// TwinCAT 3 PLC project MainPLC
// ProgramVersion: 3.1.4026.13
// libraries:
//   Tc2_BA, * (Beckhoff Automation GmbH)
//   Tc2_EtherCAT, * (Beckhoff Automation GmbH)
//   Tc2_Math, * (Beckhoff Automation GmbH)
//   Tc2_Standard, * (Beckhoff Automation GmbH)
//   Tc2_System, * (Beckhoff Automation GmbH)
//   Tc2_Utilities, * (Beckhoff Automation GmbH)
//   Tc3_EventLogger, * (Beckhoff Automation GmbH)
//   Tc3_IotBase, * (Beckhoff Automation GmbH)
// project tree:
//   DUTs/ARDeviceAPI/ keyValuePair_t.TcDUT
//   DUTs/ARDeviceErrorSystemLinker/ ARDeviceErrorSystemLink_t.TcDUT
//   DUTs/ErrorSystem/ ActorMovingTimeoutEx_t.TcDUT, ActorStartMovingtimeoutEx_t.TcDUT, IOExpantionMessageErrorEx_t.TcDUT, PrimitiveWatchdogEx_t.TcDUT
//   DUTs/IOExpantionHandler/ actorID_t.TcDUT, IOExpantionLocation_t.TcTLEO, IOExpantionMessageDescriptor_t.TcDUT, IOExpantionMessageSubData_t.TcDUT, sensorID_t.TcTLEO
//   DUTs/MainStateMachine/ mainStateMachineStatus_t.TcTLEO
//   DUTs/SignalStatusLampTypes/ SignalStatusLampStatus_t.TcTLEO
//   DUTs/systemOperationalTypes/ systemStatus_t.TcTLEO
//   GVLs/ ErrorSystemStatusVar.TcGVL, HMIInterface.TcGVL, InputOutput.TcGVL, test.TcGVL
//   / Klassendiagramm_1.TcCD (not stored), PlcTask.TcTTO
//   POUs/ARCommunication/ ARDeviceAPI_t.TcPOU, ARDeviceErrorSystemLinkerInitialiser.TcPOU, ARDeviceErrorSystemLinker_t.TcPOU
//   POUs/ARCommunication/Helper/ pulseSignalGenerator_t.TcPOU, WSJSONStringBuilder_t.TcPOU
//   POUs/ARCommunication/MQTT/ ARCommunicationMQTTExtention_t.TcPOU, ARCommunicationMQTT_t.TcPOU
//   POUs/ARCommunication/Websocket/ ARCommunicationWSExtentionWS_t.TcPOU, ARCommunicationWS_t.TcPOU
//   POUs/ARUIHandler/ ARUIHandler_t.TcPOU
//   POUs/ErrorSystem/ ActorStartMovingTimeoutManager_t.TcPOU, GernericErrorWatchdog_t.TcPOU, ActorMovingTimeoutManager_t.TcPOU, ErrorManager_t.TcPOU, formatPosition.TcPOU, IOExpantionMessageErrorHandler_t.TcPOU, PrimitiveWatchdogManager_t.TcPOU, SendErrorMessage.TcPOU
//   POUs/HMIHandler/ HMIHandler_t.TcPOU
//   POUs/IOExpantionHandler/ IOExpantionHandler_t.TcPOU
//   POUs/ MAIN.TcPOU
//   POUs/MainStateMachine/ mainStateMachine_t.TcPOU
//   POUs/SignalStatusLamp/ SignalStatusLampComponent_t.TcPOU, SignalStatusLamp_t.TcPOU
// real-time tasks:
//   TASK PlcTask: cycle T#10ms, priority 20, ADS port 350
// I/O:
//   DEVICE Gerät 1 (EtherCAT), AmsNetId 5.85.199.196.2.1
//     Klemme 1 (EK1200) [EK1200-5000 EtherCAT Netzteil (2A E-Bus)]
//       Klemme 2 (EL2869) [EL2869 16K. Dig. Ausgang 24V, 0,5A, Diagnose]
//       Klemme 3 (EL1808) [EL1808 8K. Dig. Eingang 24V, 3ms]
//       Klemme 4 (EL1808) [EL1808 8K. Dig. Eingang 24V, 3ms]
//       Klemme 5 (EL4022) [EL4022 2K. Ana. Ausgang 4-20mA, 12bit]
//       Klemme 6 (EL4104) [EL4104 4Ch. Ana. Ausgang 0-10V, 16bit]
//       Klemme 7 (EL3172) [EL3172 2K. Ana. Eingang +/-10V, +/-20mA, 16 Bit, Galvanisch getrennt]
//       Klemme 8 (EL9011) [EL9011 Endklemme]
//   DEVICE Gerät 3 (EtherCAT), AmsNetId 5.85.199.196.4.1
//     Box 9 (54632) [IMPACT67 Pro EC DIO8 IOL8]
//       modules: Module 1 (Digital_IN), Module 2 (Digital_IN), Module 3 (Digital_IN), Module 4 (Digital_IN), Module 5 (Digital_IN), Module 6 (IOL_0/4_I/O-Bytes), Module 7 (Digital_IN), Module 8 (IOL_4/4_I/O-Bytes)
// variable links:
//   MainPLC/MainPLC Instance <-> Device 1 (EtherCAT)/Term 1 (EK1200)/Term 2 (EL2869)
//     PlcTask Outputs/InputOutput.ConvaorbeltMotorReverse <-> DOS Outputs Channel 7/Output
//     PlcTask Outputs/InputOutput.ConvaorbeltMotorRun <-> DOS Outputs Channel 6/Output
//     PlcTask Outputs/InputOutput.OnOffStatusLamp <-> DOS Outputs Channel 12/Output
//     PlcTask Outputs/InputOutput.QuittierenLamp <-> DOS Outputs Channel 11/Output
//     PlcTask Outputs/InputOutput.TurnTableMotorReverse <-> DOS Outputs Channel 5/Output
//     PlcTask Outputs/InputOutput.TurnTableMotorTurn <-> DOS Outputs Channel 4/Output
//     PlcTask Outputs/MAIN.signalStatusLamp._signalLampGreen._SignalStatusLamp <-> DOS Outputs Channel 3/Output
//     PlcTask Outputs/MAIN.signalStatusLamp._signalLampRed._SignalStatusLamp <-> DOS Outputs Channel 1/Output
//     PlcTask Outputs/MAIN.signalStatusLamp._signalLampYellow._SignalStatusLamp <-> DOS Outputs Channel 2/Output
//   MainPLC/MainPLC Instance <-> Device 1 (EtherCAT)/Term 1 (EK1200)/Term 3 (EL1808)
//     PlcTask Inputs/InputOutput.EmStop <-> Channel 5/Input
//     PlcTask Inputs/InputOutput.ResetButton <-> Channel 6/Input
//   MainPLC/MainPLC Instance <-> Device 1 (EtherCAT)/Term 1 (EK1200)/Term 4 (EL1808)
//     PlcTask Inputs/InputOutput.StartButton <-> Channel 1/Input
//     PlcTask Inputs/InputOutput.StopButton <-> Channel 2/Input
//   MainPLC/MainPLC Instance <-> Device 3 (EtherCAT)/Box 9 (54632)
//     PlcTask Inputs/MAIN.IOExpantionHandler._IOExpantionExpantionInByte_{0..3} <-> Module 8 (IOL_4/4_I/O-Bytes)/TxPDO/input byte {0..3}  (4 links)
//     PlcTask Inputs/MAIN.IOExpantionHandler._IOExpantionIn_0 <-> TxPDO Mapping of Digital Inputs/PD (I/Q Pin2 + C/Q Pin4)
//     PlcTask Outputs/MAIN.IOExpantionHandler._FestoPneumaticOutByte_{0..3} <-> Module 6 (IOL_0/4_I/O-Bytes)/RxPDO/output byte {0..3}  (4 links)

CONFIGURATION MainPLC
    RESOURCE PLC ON TwinCAT3
        TASK PlcTask(INTERVAL := T#10ms, PRIORITY := 20);
        PROGRAM MAIN WITH PlcTask : MAIN;
    END_RESOURCE
END_CONFIGURATION

// ---- DUTs/ARDeviceAPI/keyValuePair_t.TcDUT
TYPE keyValuePair_t :
STRUCT
	key : STRING(255);
	value : string(255);
END_STRUCT
END_TYPE

// ---- DUTs/ARDeviceErrorSystemLinker/ARDeviceErrorSystemLink_t.TcDUT
TYPE ARDeviceErrorSystemLink_t :
STRUCT
	stEventEntity : TcEventEntry;
	callBackPtr : POINTER to bool;
END_STRUCT
END_TYPE

// ---- DUTs/ErrorSystem/ActorMovingTimeoutEx_t.TcDUT
// tis is a class that is used by the ActorMovingTimeoutManager
TYPE ActorMovingTimeoutEx_t :
STRUCT
	ActorMovingTimeout : GernericErrorWatchdog_t;
	sensorPtr1 : POINTER TO BOOL := NULL;
	sensorPtr2 : POINTER TO BOOL := NULL;
	sensorPtr3 : POINTER TO BOOL := NULL;
	sensorID1 : sensorID_t := sensorID_t.SENSOR_NO_SENSOR;
	sensorID2 : sensorID_t := sensorID_t.SENSOR_NO_SENSOR;
	sensorID3 : sensorID_t := sensorID_t.SENSOR_NO_SENSOR;
END_STRUCT
END_TYPE

// ---- DUTs/ErrorSystem/ActorStartMovingtimeoutEx_t.TcDUT
TYPE ActorStartMovingtimeoutEx_t :
STRUCT
	ActorStartMovingTimeout : GernericErrorWatchdog_t;
	expectedActorValue : BOOL; // actor value when sensor is true
	sensorPtr : POINTER TO BOOL := NULL;
	actorPtr : POINTER TO BOOL := NULL;
	sensorID : sensorID_t := sensorID_t.SENSOR_NO_SENSOR;
	actorID : actorID_t := actorID_t.ACTOR_NO_ACTOR;
END_STRUCT
END_TYPE

// ---- DUTs/ErrorSystem/IOExpantionMessageErrorEx_t.TcDUT
TYPE IOExpantionMessageErrorEx_t :
STRUCT
	isErrorActive : BOOL := FALSE; // a variable to attach to primitiveWatchdogHandler
	errorMessageCallback : BOOL := FALSE; // callback for IOExpantionHandler_t
	clearMessageCallback : BOOL := FALSE; // callback for IOExpantionHandler_t
END_STRUCT
END_TYPE

// ---- DUTs/ErrorSystem/PrimitiveWatchdogEx_t.TcDUT
TYPE PrimitiveWatchdogEx_t :
STRUCT
	primitiveWatchdog : GernericErrorWatchdog_t;
	invert : BOOL := FALSE; // if true, inverts the watchdog feeding signal
	sensorID : sensorID_t := sensorID_t.SENSOR_NO_SENSOR;
	sensorPtr : POINTER TO BOOL := NULL;
END_STRUCT
END_TYPE

// ---- DUTs/IOExpantionHandler/actorID_t.TcDUT
{attribute 'qualified_only'}
{attribute 'strict'}
{attribute 'to_string'}
TYPE actorID_t :
(
	ACTOR_0 := 0,
	ACTOR_1,
	ACTOR_2,
	ACTOR_3,
	ACTOR_GRIPPER_RIGHT_LEFT,
	ACTOR_GRIPPER_OPEN_CLOSE,
	ACTOR_GRIPPER_UP_DOWN,
	ACTOR_Y1_OUT,
	ACTOR_Y2_OUT,
	ACTOR_Y3_OUT,
	ACTOR_NO_ACTOR
);
END_TYPE

// ---- DUTs/IOExpantionHandler/IOExpantionLocation_t.TcTLEO
{attribute 'qualified_only'}
{attribute 'strict'}
{attribute 'to_string'}
TYPE IOExpantionLocation_t :
( 
	ROOT := 0, // this is the main IO master
	EXPANTION  // this is the expantion of the IO master
);
END_TYPE

// ---- DUTs/IOExpantionHandler/IOExpantionMessageDescriptor_t.TcDUT
TYPE IOExpantionMessageDescriptor_t :
STRUCT
	diagCode : ARRAY [0..3] OF BYTE;
	textID : ARRAY [0..1] OF BYTE;
END_STRUCT
END_TYPE

// ---- DUTs/IOExpantionHandler/IOExpantionMessageSubData_t.TcDUT
TYPE IOExpantionMessageSubData_t :
STRUCT
	callbackVariable : POINTER TO BOOL := NULL;
	messageDescription : IOExpantionMessageDescriptor_t;
END_STRUCT
END_TYPE

// ---- DUTs/IOExpantionHandler/sensorID_t.TcTLEO
{attribute 'qualified_only'}
{attribute 'strict'}
{attribute 'to_string'}
TYPE sensorID_t :
(
	SENSOR_B8_CONVAYORBELT_METTAL_PRESENT := 0, 
	SENSOR_B5_STORAGE_ENTRANCE,
	
	SENSOR_B17_GRIPPER_RIGHT, 
	SENSOR_B16_GRIPPER_LEFT,
	
	SENSOR_B3_Y3_DOWN, 
	SENSOR_B4_Y3_UP,
	
	EXPANTION_SENSOR_Y4_UP, 
	EXPANTION_SENSOR_B11_Y5_INSIDE,
	
	EXPANTION_SENSOR_B7_ENTRANCE_CONVAYORBELT, 
	EXPANTION_SENSOR_B6_PART_SENSOR_METTAL_PRESENT,
	
	EXPANTION_SENSOR_B12_PART_TURNTABLE_PRESENT, 
	EXPANTION_SENSOR_Y4_DOWN,
	
	EXPANTION_SENSOR_B10_Y5_OUT, 
	EXPANTION_SENSOR_B18_SENSOR_Y4,
	
	EXPANTION_SENSOR_B1_Y2_DOWN, 
	EXPANTION_SENSOR_B2_Y2_UP,
	
	SENSOR_PNEUMATIC_PRESHURE_OK,
	SENSOR_B13_TURNTABLE_POS_REACHED,
	SENSOR_NO_SENSOR
);
END_TYPE

// ---- DUTs/MainStateMachine/mainStateMachineStatus_t.TcTLEO
{attribute 'qualified_only'}
{attribute 'strict'}
{attribute 'to_string'}
TYPE mainStateMachineStatus_t :
(
	IDLE := 0,
	ROTATE_TABLE,
	GRIPPER_DOWN,
	GRIPPER_CLOSE,
	GRIPPER_UP,
	GRIPPER_LEFT,
	GRIPPER_DOWN_LEFT,
	GRIPPER_OPEN,
	GRIPPER_UP_LEFT,
	GRIPPER_RIGHT,
	Y10_OUT,
	CONVAYORBELT_START,
	Y10_BACK,
	Y2_OUT,
	Y3_OUT,
	CONVEYORBELT_STOP
);
END_TYPE

// ---- DUTs/SignalStatusLampTypes/SignalStatusLampStatus_t.TcTLEO
{attribute 'qualified_only'}
{attribute 'strict'}
{attribute 'to_string'}
TYPE SignalStatusLampStatus_t :
(
	NONE := 0,
	OPERATIONAL := 1,
	WARNING := 2,
	ERROR := 3,
	STARTING := 4,
	STOPPING := 5
);
END_TYPE

// ---- DUTs/systemOperationalTypes/systemStatus_t.TcTLEO
{attribute 'qualified_only'}
{attribute 'strict'}
{attribute 'to_string'}
TYPE systemStatus_t :
(
	STOPPED := 0,
	STARTING := 1,
	RUNNING := 2,
	ERROR := 3,
	STOPPING := 4
);
END_TYPE

// ---- GVLs/ErrorSystemStatusVar.TcGVL
{attribute 'qualified_only'}
VAR_GLOBAL
	errorHide_ERR_PNEU_LOW_PR_402 : BOOL := FALSE;
	errorHide_ERR_LD_START_LEFT_408_TIMEOUT : BOOL := FALSE;
	errorHide_ERR_LD_START_RIGHT_408_TIMEOUT : BOOL := FALSE;
	errorHide_ERR_LD_MOVE_408_TIMEOUT : BOOL := FALSE;
	errorHide_ERR_RT_MOVE_408_TIMEOUT : BOOL := FALSE;
	errorHide_ERR_Y2_MOVE_408_TIMEOUT : BOOL := FALSE;
	errorHide_ERR_Y2_START_DOWN_408_TIMEOUT : BOOL := FALSE;
	errorHide_ERR_Y2_START_UP_408_TIMEOUT : BOOL := FALSE;
	errorHide_ERR_Y3_MOVE_408_TIMEOUT : BOOL := FALSE;
	errorHide_ERR_Y3_START_DOWN_408_TIMEOUT : BOOL := FALSE;
	errorHide_ERR_Y3_START_UP_408_TIMEOUT : BOOL := FALSE;
END_VAR

// ---- GVLs/HMIInterface.TcGVL
{attribute 'qualified_only'}
VAR_GLOBAL
	HMIStartStatusLamp : BOOL := FALSE;
	HMIStopStatusLamp : BOOL := FALSE;
	HMIErrorStatusLamp : BOOL := FALSE;
	
	HMIStartMachine : BOOL := FALSE;
	HMIStopMachine : BOOL := FALSE;
END_VAR

// ---- GVLs/InputOutput.TcGVL
{attribute 'qualified_only'}
VAR_GLOBAL
	
	// outputs
	TurnTableMotorTurn AT %Q* : BOOL;
	TurnTableMotorReverse AT %Q* : BOOL;
	ConvaorbeltMotorRun AT %Q* : BOOL;
	ConvaorbeltMotorReverse AT %Q* : BOOL;
	QuittierenLamp AT %Q* : BOOL;
	OnOffStatusLamp AT %Q* : BOOL;

	// inputs
	StartButton AT %I* : BOOL;
	StopButton AT %I* : BOOL;
	EmStop AT %I* : BOOL;
	ResetButton AT %I* : BOOL;
	
	
END_VAR

// ---- GVLs/test.TcGVL
{attribute 'qualified_only'}
VAR_GLOBAL
	testBoolLinker : BOOL := FALSE;
	testBoolLinker2 : BOOL := FALSE;
END_VAR

// ---- POUs/MAIN.TcPOU
PROGRAM MAIN
VAR
signalStatusLamp : SignalStatusLamp_t;

systemStatus : systemStatus_t := systemStatus_t.STOPPED;
ARDevice : ARDeviceAPI_t;

IOExpantionHandler : IOExpantionHandler_t;

mainStateMachine : mainStateMachine_t;

ARUIHandler : ARUIHandler_t;

HMIHandler : HMIHandler_t;

ErrorManager : ErrorManager_t;

ARDeviceErrorSystemLinker : ARDeviceErrorSystemLinker_t;

_ErrorMessage : FB_TcMessage;
_tmpStr : STRING := '';

//test
firstRun : BOOL := FALSE;
run : bool := false;
callback : BOOL := FALSE;

diagCode : ARRAY[0..3] OF BYTE := [16#03, 16#E0, 16#08, 16#00];
textID : ARRAY[0..1] OF BYTE := [16#38, 16#00];

//murr test
	ReadDiag: FB_EcCoESdoRead;
	
BuffDiagMess :Array[0..39] of byte;
	xStart: BOOL;
	ReadLength: UDINT;
END_VAR

IF firstRun = FALSE THEN 
	firstRun := TRUE;
	ARDeviceErrorSystemLinkerInitialiser(ARDeviceErrorSystemLinker, ARDevice);
END_IF


// always update mainStateMachine IOExpantionahndler refferance
mainStateMachine.IOExpantionHandler := ADR(IOExpantionHandler);

ARUIHandler.ARDevice := ADR(ARDevice);
ARUIHandler.systemStatus := ADR(systemStatus);
ARUIHandler.IOExpantionHandler := ADR(IOExpantionHandler);


HMIHandler.systemStatus := ADR(systemStatus);


IF (InputOutput.StartButton OR HMIInterface.HMIStartMachine) AND NOT (systemStatus = systemStatus_t.ERROR) THEN 
	systemStatus := systemStatus_t.RUNNING; // TODO: Starting isn't implemented jet and also isn't really needed at the moment
	//ARCommunication.sendNewMessage(ADR(testStr)); // test for websocet connection
	mainStateMachine.startStateMachine(); // start state machine
	ErrorManager.startErrors();
END_IF
	
IF (NOT InputOutput.StopButton OR HMIInterface.HMIStopMachine) THEN
	mainStateMachine.stopStateMachine(); 
	systemStatus := systemStatus_t.STOPPING; 
END_IF

IF systemStatus = systemStatus_t.STOPPING AND mainStateMachine.getIsStateMachineON() = FALSE THEN
	systemStatus := systemStatus_t.STOPPED; 
	ErrorManager.stopErrors();
END_IF

// push error test
IF (NOT InputOutput.EmStop) AND systemStatus <> systemStatus_t.ERROR AND FALSE THEN 
 			_ErrorMessage.CreateEx(TC_EVENTS.OperationalErrors.EmStopPressed, 0 ); {info 'TODO: make this a alarm and not a message'}
			_ErrorMessage.ipArguments.AddString(__POUNAME());
			_tmpStr := formatPosition(__POSITION());
			_ErrorMessage.ipArguments.AddString(_tmpStr);
			_ErrorMessage.Send(0);
END_IF


IF ErrorManager.hasError() THEN
	// overwrite systemstatus to force to error state
	systemStatus := systemStatus_t.ERROR; 
	mainStateMachine.reset(); // reset StateMachine
	ErrorManager.stopErrors();
END_IF

// reset errors 
IF InputOutput.ResetButton AND systemStatus = systemStatus_t.ERROR THEN
	systemStatus := systemStatus_t.STOPPED;
	ErrorManager.confirmAll();
	InputOutput.QuittierenLamp := FALSE;
END_IF

// set lamp of quittierung
IF ErrorManager.hasError() AND systemStatus = systemStatus_t.ERROR THEN 
	InputOutput.QuittierenLamp := TRUE;
END_IF

// set maschine running lamp 
InputOutput.OnOffStatusLamp := (systemStatus = systemStatus_t.RUNNING);

CASE systemStatus OF
	systemStatus_t.STOPPED:
		signalStatusLamp.setStatus(status:=SignalStatusLampStatus_t.NONE);
		
	systemStatus_t.STARTING:
		signalStatusLamp.setStatus(status := SignalStatusLampStatus_t.STARTING);
		
	systemStatus_t.RUNNING:
		signalStatusLamp.setStatus(status:=SignalStatusLampStatus_t.OPERATIONAL);
		
	systemStatus_t.ERROR:
		signalStatusLamp.setStatus(status:=SignalStatusLampStatus_t.ERROR);
	
	systemStatus_t.STOPPING:
		signalStatusLamp.setStatus(status:=SignalStatusLampStatus_t.STOPPING);
	
END_CASE

signalStatusLamp.update();

ARDevice.update();
ARUIHandler.update();

mainStateMachine.update();

HMIHandler.update();

ARDeviceErrorSystemLinker.update();

ErrorManager.setIOExpantionHandler(ADR(IOExpantionHandler));
ErrorManager.update();

// test
{warning 'remove test'}


(*IF firstRun = FALSE AND run THEN
	firstRun := TRUE;
	
	IOExpantionHandler.subscribe(callbackVariable := ADR(callback), diagCode := diagCode, textID := textID);
END_IF

IOExpantionHandler.comUpdate();*)


// murr test
(*ReadDiag(
	sNetId:= '5.85.199.196.4.1', 
	nSlaveAddr:=1001 , 
	nSubIndex:= 2, 
	nIndex:= 16#10F3, 
	pDstBuf:= ADR(BuffDiagMess), 
	cbBufLen:= 40, 
	bExecute:=xStart , 
	tTimeout:= T#5S, 
	bBusy=> , 
	bError=> , 
	nErrId=> , 
	cbRead=>ReadLength);
*)

END_PROGRAM

// ---- POUs/SignalStatusLamp/SignalStatusLamp_t.TcPOU
FUNCTION_BLOCK SignalStatusLamp_t
VAR_INPUT
END_VAR
VAR_OUTPUT
END_VAR
VAR
	// internal store for current status value
	_status : SignalStatusLampStatus_t;
	
	// signal almps
	_signalLampGreen : SignalStatusLampComponent_t;
	_signalLampYellow : SignalStatusLampComponent_t;
	_signalLampRed : SignalStatusLampComponent_t;
	
END_VAR

METHOD setStatus : BOOL
VAR_INPUT
	status : SignalStatusLampStatus_t;
	blinking : BOOL := FALSE;
END_VAR
_status := status;

updateStatusLamp();
END_METHOD

METHOD PUBLIC update : BOOL
VAR_INPUT
END_VAR
_signalLampGreen.update();
_signalLampYellow.update();
_signalLampRed.update();
END_METHOD

METHOD PRIVATE updateStatusLamp : BOOL
VAR_INPUT
END_VAR



CASE _status OF
	SignalStatusLampStatus_t.NONE:
		_signalLampGreen.setStatus(active := FALSE);
 		_signalLampYellow.setStatus(active := FALSE);
		_signalLampRed.setStatus(active := FALSE);
		
	SignalStatusLampStatus_t.OPERATIONAL:
		_signalLampGreen.setStatus(active := TRUE);
 		_signalLampYellow.setStatus(active := FALSE);
		_signalLampRed.setStatus(active := FALSE);
		
	SignalStatusLampStatus_t.WARNING:
		_signalLampGreen.setStatus(active := FALSE);
 		_signalLampYellow.setStatus(active := TRUE);
		_signalLampRed.setStatus(active := FALSE);
		
	SignalStatusLampStatus_t.ERROR:
		_signalLampGreen.setStatus(active := FALSE);
 		_signalLampYellow.setStatus(active := FALSE);
		_signalLampRed.setStatus(active := TRUE, blinking := TRUE, timeOnMS := 200, timeOffMS := 200);
		
	SignalStatusLampStatus_t.STARTING:
		_signalLampGreen.setStatus(active := TRUE, blinking := TRUE, timeOnMS := 200, timeOffMS := 200);
 		_signalLampYellow.setStatus(active := FALSE);
		_signalLampRed.setStatus(active := FALSE);
	
	SignalStatusLampStatus_t.STOPPING:
		_signalLampGreen.setStatus(active := TRUE, blinking := TRUE, timeOnMS := 200, timeOffMS := 200);
 		_signalLampYellow.setStatus(active := FALSE);
		_signalLampRed.setStatus(active := FALSE);
	
ELSE
	// TODO: add exeption for this case (it's impossible)
	_signalLampGreen.setStatus(active := FALSE);
	_signalLampYellow.setStatus(active := TRUE, blinking := TRUE, timeOnMS := 50);
	_signalLampRed.setStatus(active := TRUE, blinking := TRUE, timeOnMS := 50, timeOffMS := 50);
END_CASE
END_METHOD

END_FUNCTION_BLOCK

// ---- POUs/SignalStatusLamp/SignalStatusLampComponent_t.TcPOU
FUNCTION_BLOCK SignalStatusLampComponent_t
VAR_INPUT
END_VAR
VAR_OUTPUT
END_VAR
VAR
	_SignalStatusLamp AT %Q* : BOOL;
	_active : BOOL := FALSE;
	_signalStatusBlink : FB_BA_Blink;
	_blinkerActive : BOOL := FALSE;
	
	_timeOnMS : UDINT;
	_timeOffMS : UDINT;
	
END_VAR

METHOD setStatus : BOOL
VAR_INPUT
	active : BOOL;
	blinking : BOOL := FALSE;
	timeOnMS : UDINT := 100;
	timeOffMS : UDINT := 100;
	
END_VAR
	_active := active;
	_blinkerActive := blinking;
	
	_timeOnMS := timeOnMS;
	_timeOffMS := timeOffMS;
	
	_signalStatusBlink.udiTiOff := timeOffMS;
	_signalStatusBlink.udiTiOn := timeOnMS;
	_signalStatusBlink.bEn := blinking;
END_METHOD

METHOD update : BOOL
VAR_INPUT
END_VAR
_signalStatusBlink();
IF _blinkerActive AND _active THEN 
	_signalStatusBlink.bEn := TRUE;
	_SignalStatusLamp := _signalStatusBlink.bQ;
ELSE 		
	_SignalStatusLamp := _active;
END_IF
END_METHOD

END_FUNCTION_BLOCK

// ---- POUs/ARCommunication/ARDeviceAPI_t.TcPOU
// supplies the active key/value for the ARDevice. This is the function that implements ARCommunication_t
FUNCTION_BLOCK ARDeviceAPI_t
VAR_INPUT
	// input varables for ARDevice
	lmpRunning : BOOL := FALSE; // true when mashine is running
	lmpStopped : BOOL := TRUE; // true when machine is stopped
	lmpError : BOOL := FALSE; // true when machine has an error
	
	displayEMStop : BOOL := FALSE; // true when EM-Stopp (please relese) message is displayed on the controlpannel
	displayQuittierung : BOOL := FALSE; // true when Please Press me (Quittierung) is displayed on the controlpannel
	
	PneumaticOkB20_sensorStatus : BOOL := FALSE; 
	PartTurntablePresentB12_sensorStatus : BOOL := FALSE;
	LinearActuatorLeftB16_sensorStatus : BOOL := FALSE;
	LinearActuatorRightB17_sensorStatus : BOOL := FALSE;
	TurntablePositionReachedB13_sensorStatus : BOOL := FALSE;
	StorageEntranceB5_sensorStatus : BOOL := FALSE;
	ConveyorBeltMetalPresentB8_sensorStatus : BOOL := FALSE;
	EntranceConveyorBeltB7_sensorStatus : BOOL := FALSE;
	SensorPartMetalPresentB6_sensorStatus : BOOL := FALSE;
	
	errorHide_ERR_PNEU_LOW_PR_402 : BOOL := FALSE;
	errorHide_ERR_LD_START_LEFT_408_TIMEOUT : BOOL := FALSE;
	errorHide_ERR_LD_START_RIGHT_408_TIMEOUT : BOOL := FALSE;
	errorHide_ERR_LD_MOVE_408_TIMEOUT : BOOL := FALSE;
	errorHide_ERR_RT_MOVE_408_TIMEOUT : BOOL := FALSE;
	errorHide_ERR_Y2_MOVE_408_TIMEOUT : BOOL := FALSE;
	errorHide_ERR_Y2_START_DOWN_408_TIMEOUT : BOOL := FALSE;
	errorHide_ERR_Y2_START_UP_408_TIMEOUT : BOOL := FALSE;
	errorHide_ERR_Y3_MOVE_408_TIMEOUT : BOOL := FALSE;
	errorHide_ERR_Y3_START_DOWN_408_TIMEOUT : BOOL := FALSE;
	errorHide_ERR_Y3_START_UP_408_TIMEOUT : BOOL := FALSE;
	
END_VAR
VAR_OUTPUT
	// output variables from ARDevice	
	testOut : BOOL := FALSE;
END_VAR
VAR
	// sent input (to notice changes in state)	(Inifficiant as hell with more parametewrs but who cares)
	_lmpRunning : BOOL := FALSE; // true when mashine is running
	_lmpStopped : BOOL := TRUE; // true when machine is stopped
	_lmpError : BOOL := FALSE; // true when machine has an error

	_displayEMStop : BOOL := FALSE; // true when EM-Stopp (please relese) message is displayed on the controlpannel
	_displayQuittierung : BOOL := FALSE; // true when Please Press me (Quittierung) is displayed on the controlpannel

	_PneumaticOkB20_sensorStatus : BOOL := FALSE; 
	_PartTurntablePresentB12_sensorStatus : BOOL := FALSE;
	_LinearActuatorLeftB16_sensorStatus : BOOL := FALSE;
	_LinearActuatorRightB17_sensorStatus : BOOL := FALSE;
	_TurntablePositionReachedB13_sensorStatus : BOOL := FALSE;
	_StorageEntranceB5_sensorStatus : BOOL := FALSE;
	_ConveyorBeltMetalPresentB8_sensorStatus : BOOL := FALSE;
	_EntranceConveyorBeltB7_sensorStatus : BOOL := FALSE;
	_SensorPartMetalPresentB6_sensorStatus : BOOL := FALSE;

	_errorHide_ERR_PNEU_LOW_PR_402 : BOOL := FALSE;
	_errorHide_ERR_LD_START_LEFT_408_TIMEOUT : BOOL := FALSE;
	_errorHide_ERR_LD_START_RIGHT_408_TIMEOUT : BOOL := FALSE;
	_errorHide_ERR_LD_MOVE_408_TIMEOUT : BOOL := FALSE;
	_errorHide_ERR_RT_MOVE_408_TIMEOUT : BOOL := FALSE;
	_errorHide_ERR_Y2_MOVE_408_TIMEOUT : BOOL := FALSE;
	_errorHide_ERR_Y2_START_DOWN_408_TIMEOUT : BOOL := FALSE;
	_errorHide_ERR_Y2_START_UP_408_TIMEOUT : BOOL := FALSE;
	_errorHide_ERR_Y3_MOVE_408_TIMEOUT : BOOL := FALSE;
	_errorHide_ERR_Y3_START_DOWN_408_TIMEOUT : BOOL := FALSE;
	_errorHide_ERR_Y3_START_UP_408_TIMEOUT : BOOL := FALSE;

	_ARCommunication : ARCommunicationMQTT_t;
	_WSRequestBiuilder : WSJSONStringBuilder_t;
	_reSendSignal : pulseSignalGenerator_t;
END_VAR

// for adding a new in value:
// 		add variable in VAR_INPUT
//		add variable in VAR
// 		add in sendData an attribute
// 		add in sendData an update from the VAR_INPUT variable to the VAR variable
//		add detect new state in detectNewState
//
// for adding a new out value
// 		add variable in VAR_OUTPUT
// 		add if statement in checkKeyValue and update VAR_OUT value

// this is for intreperting the values from the ARDevice
METHOD PRIVATE checkKeyValue : BOOL
VAR_INPUT
	keyValuePair : keyValuePair_t;
END_VAR

IF keyValuePair.key = 'testOut'THEN
	testOut := ConvertToBool(keyValuePair.value);
ELSE
	; // no other outputs
END_IF;
END_METHOD

METHOD PRIVATE ConvertToBool : BOOL
VAR_INPUT
	str : string(255);
END_VAR
str := delete(str, 1, 1);
str := delete(str, 1, len(str));
ConvertToBool := STRING_TO_BOOL(str);
return;
END_METHOD

// this class is for deconstructiong a message form ARDevice (if the ARDeviuce sends more than 50 key/value paris, this function cannot handle that)
METHOD PRIVATE deconstructMessage : BOOL
VAR_INPUT
	message : STRING(255);
END_VAR
VAR
	_buffer : ARRAY [0..50] OF keyValuePair_t;
	
	i : UINT := 0;
	_activeKeyValuePair : keyValuePair_t;
	_activeValueTokenPair : STRING(255) := '';
	_ValTokenPairDelimitorIndex : INT := 0; // ','
	_ValTokenDelimitorIndex : INT := 0; // ':'
END_VAR
IF message = 'ERROR' THEN
	{info 'TODO: Implement error handeling for this case (throw a warning or something)'}
	deconstructMessage := FALSE;
	RETURN;
END_IF

IF len(message) < 2 THEN 
	{info 'TODO: Implement error handeling for this case (throw a warning or something)'}
	deconstructMessage := FALSE;
	RETURN;
END_IF

// remove '{' and '}' (no, i'm not processing the JSON String prperly, but who cares) 
message := delete(message, 1, 1);
message := delete(message, 1, len(message));

WHILE len(message) <> 0 DO
	// extract token
	_ValTokenPairDelimitorIndex := find(message, ',');
	IF _ValTokenPairDelimitorIndex = 0 THEN // last token
		_activeValueTokenPair := message;
		message := ''; 
	ELSE // not last token
		_activeValueTokenPair := left(message, _ValTokenPairDelimitorIndex - 1); 
		message := delete(message, _ValTokenPairDelimitorIndex, 1);
	END_IF
	
	// extract key and value out of key value pair
	_ValTokenDelimitorIndex := find(_activeValueTokenPair, ':');
	
	IF(_ValTokenDelimitorIndex = 0) THEN // wut?
		{info: 'trow a warning and drop packet, something is wrong'}
		deconstructMessage := FALSE;
		RETURN;
	END_IF
	
	_activeKeyValuePair.key := left(_activeValueTokenPair, _valTokenDelimitorIndex - 1);
	_activeValueTokenPair := delete(_activeValueTokenPair, _valTokenDelimitorIndex, 1);
	_activeKeyValuePair.value := _activeValueTokenPair;
	
	_activeKeyValuePair.key := delete(_activeKeyValuePair.key, 1, 1);
	_activeKeyValuePair.key := delete(_activeKeyValuePair.key, 1, len(_activeKeyValuePair.key));
	
	_buffer[i] := _activeKeyValuePair;
	
	i := i + 1;
END_WHILE

// interprete every value
FOR i := 0 TO 50 DO
	IF _buffer[i].key = '' THEN // end of buffer reached
		deconstructMessage := TRUE;
		RETURN;
	END_IF
	checkKeyValue(_buffer[i]);	// parse and set out variable
END_FOR

RETURN;
END_METHOD

METHOD PRIVATE detectNewState : BOOL
VAR_INPUT
END_VAR
// list all in parameters here
detectNewState := detectNewState OR (_lmpRunning XOR lmpRunning);
detectNewState := detectNewState OR (_lmpStopped XOR lmpStopped);
detectNewState := detectNewState OR (_lmpError XOR lmpError);

detectNewState := detectNewState OR (_displayEMStop XOR displayEMStop);
detectNewState := detectNewState OR (_displayQuittierung XOR displayQuittierung);

detectNewState := detectNewState OR (_PneumaticOkB20_sensorStatus XOR PneumaticOkB20_sensorStatus);
detectNewState := detectNewState OR (_PartTurntablePresentB12_sensorStatus XOR PartTurntablePresentB12_sensorStatus);
detectNewState := detectNewState OR (_LinearActuatorLeftB16_sensorStatus XOR LinearActuatorLeftB16_sensorStatus);
detectNewState := detectNewState OR (_LinearActuatorRightB17_sensorStatus XOR LinearActuatorRightB17_sensorStatus);
detectNewState := detectNewState OR (_TurntablePositionReachedB13_sensorStatus XOR TurntablePositionReachedB13_sensorStatus);
detectNewState := detectNewState OR (_StorageEntranceB5_sensorStatus XOR StorageEntranceB5_sensorStatus);
detectNewState := detectNewState OR (_ConveyorBeltMetalPresentB8_sensorStatus XOR ConveyorBeltMetalPresentB8_sensorStatus);
detectNewState := detectNewState OR (_EntranceConveyorBeltB7_sensorStatus XOR EntranceConveyorBeltB7_sensorStatus);
detectNewState := detectNewState OR (_SensorPartMetalPresentB6_sensorStatus XOR SensorPartMetalPresentB6_sensorStatus);

detectNewState := detectNewState OR (_errorHide_ERR_PNEU_LOW_PR_402 XOR errorHide_ERR_PNEU_LOW_PR_402);
detectNewState := detectNewState OR (_errorHide_ERR_LD_START_LEFT_408_TIMEOUT XOR errorHide_ERR_LD_START_LEFT_408_TIMEOUT);
detectNewState := detectNewState OR (_errorHide_ERR_LD_START_RIGHT_408_TIMEOUT XOR errorHide_ERR_LD_START_RIGHT_408_TIMEOUT);
detectNewState := detectNewState OR (_errorHide_ERR_LD_MOVE_408_TIMEOUT XOR errorHide_ERR_LD_MOVE_408_TIMEOUT);
detectNewState := detectNewState OR (_errorHide_ERR_RT_MOVE_408_TIMEOUT XOR errorHide_ERR_RT_MOVE_408_TIMEOUT);
detectNewState := detectNewState OR (_errorHide_ERR_Y2_MOVE_408_TIMEOUT XOR errorHide_ERR_Y2_MOVE_408_TIMEOUT);
detectNewState := detectNewState OR (_errorHide_ERR_Y2_START_DOWN_408_TIMEOUT XOR errorHide_ERR_Y2_START_DOWN_408_TIMEOUT);
detectNewState := detectNewState OR (_errorHide_ERR_Y2_START_UP_408_TIMEOUT XOR errorHide_ERR_Y2_START_UP_408_TIMEOUT);
detectNewState := detectNewState OR (_errorHide_ERR_Y3_MOVE_408_TIMEOUT XOR errorHide_ERR_Y3_MOVE_408_TIMEOUT);
detectNewState := detectNewState OR (_errorHide_ERR_Y3_START_DOWN_408_TIMEOUT XOR errorHide_ERR_Y3_START_DOWN_408_TIMEOUT);
detectNewState := detectNewState OR (_errorHide_ERR_Y3_START_UP_408_TIMEOUT XOR errorHide_ERR_Y3_START_UP_408_TIMEOUT);

return;
END_METHOD

// sends whole state to ARDevice
METHOD PRIVATE sendData : BOOL
VAR_INPUT
END_VAR
// build syntax
_WSRequestBiuilder.clear();

// add  attributes
_WSRequestBiuilder.addAttributeBool('lmpRunning', lmpRunning);
_WSRequestBiuilder.addAttributeBool('lmpStopped', lmpStopped);
_WSRequestBiuilder.addAttributeBool('lmpError', lmpError);

_WSRequestBiuilder.addAttributeBool('displayEMStop', displayEMStop);
_WSRequestBiuilder.addAttributeBool('displayQuittierung', displayQuittierung);

_WSRequestBiuilder.addAttributeBool('PneumaticOkB20_sensorStatus', PneumaticOkB20_sensorStatus);
_WSRequestBiuilder.addAttributeBool('PartTurntablePresentB12_sensorStatus', PartTurntablePresentB12_sensorStatus);
_WSRequestBiuilder.addAttributeBool('LinearActuatorLeftB16_sensorStatus', LinearActuatorLeftB16_sensorStatus);
_WSRequestBiuilder.addAttributeBool('LinearActuatorRightB17_sensorStatus', LinearActuatorRightB17_sensorStatus);
_WSRequestBiuilder.addAttributeBool('TurntablePositionReachedB13_sensorStatus', TurntablePositionReachedB13_sensorStatus);
_WSRequestBiuilder.addAttributeBool('StorageEntranceB5_sensorStatus', StorageEntranceB5_sensorStatus);
_WSRequestBiuilder.addAttributeBool('ConveyorBeltMetalPresentB8_sensorStatus', ConveyorBeltMetalPresentB8_sensorStatus);
_WSRequestBiuilder.addAttributeBool('EntranceConveyorBeltB7_sensorStatus', EntranceConveyorBeltB7_sensorStatus);
_WSRequestBiuilder.addAttributeBool('SensorPartMetalPresentB6_sensorStatus', SensorPartMetalPresentB6_sensorStatus);

_WSRequestBiuilder.addAttributeBool('ERR_PNEU_LOW_PR_402', errorHide_ERR_PNEU_LOW_PR_402);
_WSRequestBiuilder.addAttributeBool('ERR_LD_START_LEFT_408_TIMEOUT', errorHide_ERR_LD_START_LEFT_408_TIMEOUT);
_WSRequestBiuilder.addAttributeBool('ERR_LD_START_RIGHT_408_TIMEOUT', errorHide_ERR_LD_START_RIGHT_408_TIMEOUT);
_WSRequestBiuilder.addAttributeBool('ERR_LD_MOVE_408_TIMEOUT', errorHide_ERR_LD_MOVE_408_TIMEOUT);
_WSRequestBiuilder.addAttributeBool('ERR_RT_MOVE_408_TIMEOUT', errorHide_ERR_RT_MOVE_408_TIMEOUT);
_WSRequestBiuilder.addAttributeBool('ERR_Y2_MOVE_408_TIMEOUT', errorHide_ERR_Y2_MOVE_408_TIMEOUT);
_WSRequestBiuilder.addAttributeBool('ERR_Y2_START_DOWN_408_TIMEOUT', errorHide_ERR_Y2_START_DOWN_408_TIMEOUT);
_WSRequestBiuilder.addAttributeBool('ERR_Y2_START_UP_408_TIMEOUT', errorHide_ERR_Y2_START_UP_408_TIMEOUT);
_WSRequestBiuilder.addAttributeBool('ERR_Y3_MOVE_408_TIMEOUT', errorHide_ERR_Y3_MOVE_408_TIMEOUT);
_WSRequestBiuilder.addAttributeBool('ERR_Y3_START_DOWN_408_TIMEOUT', errorHide_ERR_Y3_START_DOWN_408_TIMEOUT);
_WSRequestBiuilder.addAttributeBool('ERR_Y3_START_UP_408_TIMEOUT', errorHide_ERR_Y3_START_UP_408_TIMEOUT);


// update states 
_lmpRunning := lmpRunning;
_lmpStopped := lmpStopped;
_lmpError := lmpError;


_PneumaticOkB20_sensorStatus := PneumaticOkB20_sensorStatus;
_PartTurntablePresentB12_sensorStatus := PartTurntablePresentB12_sensorStatus;
_LinearActuatorLeftB16_sensorStatus := LinearActuatorLeftB16_sensorStatus;
_LinearActuatorRightB17_sensorStatus := LinearActuatorRightB17_sensorStatus;
_TurntablePositionReachedB13_sensorStatus := TurntablePositionReachedB13_sensorStatus;
_StorageEntranceB5_sensorStatus := StorageEntranceB5_sensorStatus;
_ConveyorBeltMetalPresentB8_sensorStatus := ConveyorBeltMetalPresentB8_sensorStatus;
_EntranceConveyorBeltB7_sensorStatus := EntranceConveyorBeltB7_sensorStatus;
_SensorPartMetalPresentB6_sensorStatus := SensorPartMetalPresentB6_sensorStatus;

_errorHide_ERR_PNEU_LOW_PR_402 := errorHide_ERR_PNEU_LOW_PR_402;
_errorHide_ERR_LD_START_LEFT_408_TIMEOUT := errorHide_ERR_LD_START_LEFT_408_TIMEOUT;
_errorHide_ERR_LD_START_RIGHT_408_TIMEOUT := errorHide_ERR_LD_START_RIGHT_408_TIMEOUT;
_errorHide_ERR_LD_MOVE_408_TIMEOUT := errorHide_ERR_LD_MOVE_408_TIMEOUT;
_errorHide_ERR_RT_MOVE_408_TIMEOUT := errorHide_ERR_RT_MOVE_408_TIMEOUT;
_errorHide_ERR_Y2_MOVE_408_TIMEOUT := errorHide_ERR_Y2_MOVE_408_TIMEOUT;
_errorHide_ERR_Y2_START_DOWN_408_TIMEOUT := errorHide_ERR_Y2_START_DOWN_408_TIMEOUT;
_errorHide_ERR_Y2_START_UP_408_TIMEOUT := errorHide_ERR_Y2_START_UP_408_TIMEOUT;
_errorHide_ERR_Y3_MOVE_408_TIMEOUT := errorHide_ERR_Y3_MOVE_408_TIMEOUT;
_errorHide_ERR_Y3_START_DOWN_408_TIMEOUT := errorHide_ERR_Y3_START_DOWN_408_TIMEOUT;
_errorHide_ERR_Y3_START_UP_408_TIMEOUT := errorHide_ERR_Y3_START_UP_408_TIMEOUT;


_displayEMStop := displayEMStop;
_displayQuittierung := displayQuittierung;

//build and send
_ARCommunication.sendNewMessage(_WSRequestBiuilder.build());
END_METHOD

// must be called as oftern as possible if it returns false, something is wrong with the sending or reciving attribute
METHOD update : BOOL
VAR_INPUT
END_VAR
VAR
	test : bool := false;
END_VAR
_ARCommunication.update();
_reSendSignal.update();

IF _ARCommunication.getConnectionStatus() = FALSE THEN
	return;
END_IF

// check for changes to send
IF detectNewState() OR _reSendSignal.signal  THEN
	sendData();
END_IF

// check for new messages
IF _ARCommunication.newMessageRecived() THEN
	deconstructMessage(_ARCommunication.getLastMessage());
END_IF
END_METHOD

END_FUNCTION_BLOCK

// ---- POUs/ARCommunication/MQTT/ARCommunicationMQTT_t.TcPOU
FUNCTION_BLOCK ARCommunicationMQTT_t
VAR_INPUT
END_VAR
VAR_OUTPUT
END_VAR
VAR
	_CommunicationImplementation : ARCommunicationMQTTExtention_t;
	_publishTopic : STRING(255) := 'PLC'; 
	_subscribeTopic : STRING(255) := 'ARDevice';
	
	
	_SetParameter : BOOL := TRUE;
	_Connect : BOOL := TRUE;
	_errorOccured : HRESULT;
	_Subscribed : bool := false;
END_VAR

METHOD getConnectionStatus : BOOL
VAR_INPUT
END_VAR
getConnectionStatus := _CommunicationImplementation.bConnected;
return;
END_METHOD

METHOD getLastMessage : STRING(255)
VAR_INPUT
END_VAR
getLastMessage := _CommunicationImplementation.getPayload();
_CommunicationImplementation.newMessageAvalable := false;
END_METHOD

METHOD newMessageRecived : BOOL
VAR_INPUT
END_VAR
newMessageRecived := _CommunicationImplementation.newMessageAvalable;
END_METHOD

METHOD sendNewMessage : BOOL
VAR_INPUT
	str : STRING(2000); // (max str length 2000)
END_VAR

VAR
END_VAR
_CommunicationImplementation.Publish(sTopic := _publishTopic, pPayload := ADR(str), nPayloadSize := Len2(ADR(str))+1);

IF _CommunicationImplementation.bError THEN
	sendNewMessage := FALSE;
	RETURN;
END_IF

sendNewMessage := TRUE;
return;
END_METHOD

METHOD update : BOOL
VAR_INPUT
END_VAR
IF _SetParameter THEN
	_SetParameter := FALSE;
	_CommunicationImplementation.sHostName:= 'localhost';
	_CommunicationImplementation.nHostPort:= 1883;
//	_CommunicationImplementation.sClientId:= 'MyTcMqttClient'; 
	_CommunicationImplementation.sTopicPrefix:= ''; 
//	_CommunicationImplementation.nKeepAlive:= 60; 
//	_CommunicationImplementation.sUserName:= ;
//	_CommunicationImplementation.sUserPassword:= ; 
//	_CommunicationImplementation.stWill:= ; 
//	_CommunicationImplementation.stTLS:= ;
END_IF

_CommunicationImplementation.Execute(_Connect);
IF _CommunicationImplementation.bError THEN
	// add your error logging here
	_errorOccured := _CommunicationImplementation.hrErrorCode;
END_IF

IF _CommunicationImplementation.bConnected THEN
	IF NOT _Subscribed THEN
		_Subscribed := _CommunicationImplementation.Subscribe(sTopic:=_subscribeTopic, eQoS:=TcIotMqttQos.AtMostOnceDelivery);
		IF _CommunicationImplementation.bError THEN
			// add your error logging here
			_errorOccured := _CommunicationImplementation.hrErrorCode;
		END_IF
	END_IF
END_IF
END_METHOD

END_FUNCTION_BLOCK

// ---- POUs/ARCommunication/MQTT/ARCommunicationMQTTExtention_t.TcPOU
{attribute 'c++_compatible'} 
FUNCTION_BLOCK ARCommunicationMQTTExtention_t EXTENDS FB_IotMqttClient
VAR_INPUT
END_VAR
VAR_OUTPUT
END_VAR

VAR
	_newMessageAvalable : BOOL := FALSE;	

	(* received message *)
	{attribute 'TcEncoding':='UTF-8'}
	sTopicRcv : STRING(255);
	{attribute 'TcEncoding':='UTF-8'}
	sPayloadRcv : STRING(255);
END_VAR

METHOD getPayload : STRING(255)
{attribute 'c++_compatible'}
VAR_INPUT
END_VAR
getPayload := sPayloadRcv;
return;
END_METHOD

PROPERTY newMessageAvalable : BOOL
{attribute 'c++_compatible'}
GET
{attribute 'c++_compatible'}
VAR
END_VAR
newMessageAvalable := _newMessageAvalable;
return;
END_GET
SET
{attribute 'c++_compatible'}
VAR
END_VAR
_newMessageAvalable := newMessageAvalable;
return;
END_SET
END_PROPERTY

{attribute 'c++_compatible'}
{attribute 'pack_mode' := '4'}
{attribute 'show'}
{attribute 'minimal_input_size' := '4'}
METHOD OnMqttMessage : Tc3_IotBase.HRESULT
VAR_IN_OUT CONSTANT
	topic	: STRING;
END_VAR
VAR_INPUT
	(* pointer to payload*)
	payload	: Tc3_IotBase.PVOID;
	(* payload size in bytes*)
	length	: UDINT;
	qos	: Tc3_IotBase.TcIotMqttQos;
	repeated	: BOOL;
END_VAR

VAR
	nPayloadRcvLen : UDINT;
END_VAR
SUPER^.nMessagesRcv := SUPER^.nMessagesRcv + 1;

STRNCPY( ADR(sTopicRcv), ADR(topic), SIZEOF(sTopicRcv) );
nPayloadRcvLen := MIN(length, DINT_TO_UDINT(SIZEOF(sPayloadRcv))-1);
MEMCPY( ADR(sPayloadRcv), payload, nPayloadRcvLen );
sPayloadRcv[nPayloadRcvLen] := 0;  // ensure a null termination of received string

OnMqttMessage := S_OK;

_newMessageAvalable := TRUE;
END_METHOD

END_FUNCTION_BLOCK

// ---- POUs/ARCommunication/Helper/WSJSONStringBuilder_t.TcPOU
// this class is following the OOP Desgn Pattern of a builder (max str length 255)
FUNCTION_BLOCK WSJSONStringBuilder_t
VAR_INPUT
END_VAR
VAR_OUTPUT
END_VAR
VAR
	_str : STRING(2000) := '';
END_VAR

METHOD addAttributeBool : BOOL
VAR_INPUT
	key : STRING(255);
	value : BOOL;
END_VAR
addAttributeBool := addAttributeString(key, BOOL_TO_STRING(value));
return;
END_METHOD

METHOD addAttributeINT : BOOL
VAR_INPUT
	key: STRING(255);
	value: INT;
END_VAR
VAR
	_keyValuePair: STRING(255);
	_tmpStr: STRING(255);
END_VAR
_keyValuePair := formateAttributeINT(key, value);

IF  _keyValuePair = 'ERROR' OR len(_str) + len(_keyValuePair) + 2 > 2000 THEN // length of existing string + new keyValuePar + '{' + '}'
	addAttributeINT := FALSE; 
	RETURN;
END_IF

_tmpStr := concat(_keyValuePair, ',');
concat2(ADR(_str), ADR(_tmpStr), ADR(_str), 2000); // apped key value pair to string with ',' at the end
//_str := concat(_str, concat(_keyValuePair, ',')); // apped key value pair to string with ',' at the end

addAttributeINT := TRUE;
RETURN;
END_METHOD

// adds an attribute (if it returns true: succsess, if false: failed)
METHOD addAttributeString : BOOL
VAR_INPUT
	key : STRING(255);
	value : STRING(255);
END_VAR
VAR
	_tmpStr : STRING := '';
	_keyValuePair : STRING := '';
END_VAR
_keyValuePair := formateAttribute(key, value);

IF  _keyValuePair = 'ERROR' OR len(_str) + len(_keyValuePair) + 2 > 2000 THEN // length of existing string + new keyValuePar + '{' + '}'
	addAttributeString := FALSE; 
	RETURN;
END_IF

_tmpStr := concat(_keyValuePair, ',');
concat2(ADR(_str), ADR(_tmpStr), ADR(_str), 2000); // apped key value pair to string with ',' at the end
//_str := concat(_str, concat(_keyValuePair, ',')); 

addAttributeString := TRUE;
RETURN;
END_METHOD

// builds the JSON string (if it fails output = 'ERROR')
METHOD build : STRING(1000)
VAR_INPUT
END_VAR
VAR
	_lastCharOfStr : STRING(1) := '';
	_appendStr : STRING(1) := '}';
	_prefixStr : STRING(1) := '{';
END_VAR
IF len(_str) + 1 > 2000 OR _str = '' THEN // validate data
	build := 'ERROR';
	RETURN;
END_IF

//_lastCharOfStr := right(_str, 1);

//IF _lastCharOfStr = ',' THEN // check if last character is a ','
delete2(ADR(_str), ADR(_str), 2000, 1, len2(ADR(_str)));
	//_str := delete(_str, 1, len(_str));
//END_IF

// wrap key value pair list

CONCAT2(ADR(_prefixStr), ADR(_str), ADR(_str), 2000); 
CONCAT2(ADR(_str), ADR(_appendStr), ADR(build), 2000); 
//build := concat('{', concat(_str, '}'));
RETURN;
END_METHOD

// clears whole attribute buffer
METHOD clear : BOOL
VAR_INPUT
END_VAR
_str := '';
END_METHOD

// takes a key and attribute and formats it to a valid key value pair (if string is too long ouput will be 'ERROR')
METHOD PRIVATE formateAttribute : string(255)
VAR_INPUT
	key : STRING(255);
	value : STRING(255);
END_VAR
VAR
	_tmpStr : STRING(255) := '';
END_VAR
IF LEN(key) + len(value) + 5 > 2000  THEN // return error if string is too long
	formateAttribute := 'ERROR';
	RETURN;
END_IF

// formate key value pair
_tmpStr := concat('"', key);
_tmpStr := concat(_tmpStr, '":"');
_tmpStr := concat(_tmpStr, value);
formateAttribute := concat(_tmpStr, '"');
RETURN;
END_METHOD

METHOD PRIVATE formateAttributeINT : string(255)
VAR_INPUT
	key: STRING(255);
	value: INT;
END_VAR

VAR
	_tmpStr: STRING(255);
END_VAR
IF LEN(key) + len(INT_TO_STRING(value)) + 3 > 2000  THEN // return error if string is too long
	formateAttributeINT := 'ERROR';
	RETURN;
END_IF

// formate key value pair
_tmpStr := concat('"', key);
_tmpStr := concat(_tmpStr, '":');
formateAttributeINT := concat(_tmpStr, INT_TO_STRING(value));
RETURN;
END_METHOD

END_FUNCTION_BLOCK

// ---- POUs/ARCommunication/Helper/pulseSignalGenerator_t.TcPOU
FUNCTION_BLOCK pulseSignalGenerator_t
VAR_INPUT
	durrationBetweenSignals_ms : UDINT := 10000; 
END_VAR
VAR_OUTPUT
	signal : BOOL;
END_VAR
VAR
	_timer : FB_BA_Blink;
	_state : BOOL := FALSE; 
END_VAR

METHOD update : BOOL
VAR_INPUT
END_VAR
_timer.bEn := TRUE;
_timer.udiTiOff := durrationBetweenSignals_ms;
_timer.udiTiOn := 1; 

_timer();
signal := FALSE;
IF _timer.bQ = TRUE AND _state = FALSE THEN
	_state := TRUE;
	signal := TRUE;
END_IF

IF _timer.bQ = FALSE AND _state = TRUE THEN
	_state := FALSE;
END_IF
END_METHOD

END_FUNCTION_BLOCK

// ---- POUs/IOExpantionHandler/IOExpantionHandler_t.TcPOU
FUNCTION_BLOCK IOExpantionHandler_t
VAR_INPUT
END_VAR
VAR_OUTPUT
END_VAR
VAR
 
	_IOExpantionExpantionInByte_0 AT %I* : BYTE; // in byte 0
	_IOExpantionExpantionInByte_1 AT %I* : BYTE; // in byte 1
	_IOExpantionExpantionInByte_2 AT %I* : BYTE; // diagnostic byte 2
	_IOExpantionExpantionInByte_3 AT %I* : BYTE; // user specifyed content 3
	
	_IOExpantionExpantionInBytes : ARRAY [0..3] OF POINTER TO BYTE := [ADR(_IOExpantionExpantionInByte_0), ADR(_IOExpantionExpantionInByte_1), ADR(_IOExpantionExpantionInByte_2), ADR(_IOExpantionExpantionInByte_3)];
	 
	_FestoPneumaticOutByte_0 AT %Q* : BYTE;
	_FestoPneumaticOutByte_1 AT %Q* : BYTE;
	_FestoPneumaticOutByte_2 AT %Q* : BYTE;
	_FestoPneumaticOutByte_3 AT %Q* : BYTE;
	
	_FestoPneumaticOutBytes : ARRAY [0..3] OF POINTER TO BYTE := [ADR(_FestoPneumaticOutByte_0), ADR(_FestoPneumaticOutByte_1), ADR(_FestoPneumaticOutByte_2), ADR(_FestoPneumaticOutByte_3)];
	
	_IOExpantionIn_0 AT %I* : UINT; // this input does only have two active bits (bit 0 and bit 1)
	
	_IOExpantionInBytes : ARRAY [0..0] OF POINTER TO UINT := [ADR(_IOExpantionIn_0)];
	
	_ErrorMessage : FB_TcMessage;
	
	//------------------------------------
	
	_lastMessageRead : UINT := 0; // last message retrived by this^.getNewMessage();
	_newestMessageInBuffer : UINT := 0; // newest message in ring buffer (actual newest message)
	_currentMessageRead : BYTE := 16#00; // current message being read
	
	_subscriberArray : ARRAY[0..99] OF IOExpantionMessageSubData_t;
	
	_readDiagIndex : FB_EcCoESdoRead;
	_readDiagMessage : FB_EcCoESdoRead;
	
	_readDiagMessageClock : pulseSignalGenerator_t;
	
	_returnDiagBuffer : ARRAY[0..236] OF BYTE;
	_returnIndexBuff : ARRAY[0..39] OF BYTE;
END_VAR

// this is for handeling the IO link master from murr. This is a highly specialised class that needs to be changed acording to the inputs on the expantion of IO link master from murr.

METHOD PRIVATE callCallback : BOOL
VAR_INPUT
	messageDescription : IOExpantionMessageDescriptor_t;
END_VAR
VAR
	i : UINt := 0;
END_VAR

// search for callback to call

FOR i := 0 TO TO_UINT(SIZEOF(_subscriberArray) / SIZEOF(IOExpantionMessageSubData_t)) DO
	IF isMesDesEqual(_subscriberArray[i].messageDescription, messageDescription) THEN
		IF _subscriberArray[i].callbackVariable <> NULL THEN
			_subscriberArray[i].callbackVariable^ := TRUE;
		END_IF
	END_IF
END_FOR

callCallback := TRUE;
return;
END_METHOD

// communication Update, call this every cycle
METHOD comUpdate : BOOL
VAR_INPUT
END_VAR
VAR 
	getNewestMessageIndexBusy : BOOL := FALSE;
	NewestMessageAvalableTmpOut : BYTE := 16#00;
	
	getMessageBusy : BOOL := FALSE;
END_VAR
// check if a new message is avalable
IF _newestMessageInBuffer = _lastMessageRead THEN
	NewestMessageAvalableTmpOut := getNewestMessageIndex(busy => getNewestMessageIndexBusy);
	IF getNewestMessageIndexBusy THEN
	RETURN;
	ELSE 
	_newestMessageInBuffer := NewestMessageAvalableTmpOut;
	RETURN;
	END_IF
END_IF

// read messages 
IF _readDiagMessageClock.signal THEN
	getMessage(index := _currentMessageRead, busy => getMessageBusy);
END_IF

IF getMessageBusy = FALSE THEN
	_currentMessageRead := getNextMessageIndex(_currentMessageRead);
	
	IF _currentMessageRead = _newestMessageInBuffer + 1 THEN
		_lastMessageRead := _newestMessageInBuffer;
	END_IF
	
	callCallback(genMessageDescription(ADR(_returnDiagBuffer)));
END_IF

_readDiagMessageClock.update();
END_METHOD

METHOD PRIVATE convertByteBit : BOOL
VAR_INPUT
	byteVal : BYTE;
	offset : UINT;
END_VAR

VAR
	_tmpStr: STRING;
END_VAR
IF offset > 7 THEN 
	convertByteBit := FALSE; 
	_ErrorMessage.CreateEx(TC_EVENTS.ProgrammingErrors.invalidAccsessOfBitInByte, 0 );
	_ErrorMessage.ipArguments.AddString(__POUNAME());
	_tmpStr := formatPosition(__POSITION());
	_ErrorMessage.ipArguments.AddString(_tmpStr);
	_ErrorMessage.Send(0);
	RETURN;
END_IF

convertByteBit := TO_BOOL(( byteVal AND (SHL(1, offset ))));

RETURN;
END_METHOD

METHOD PRIVATE extractSensorBit : BOOL
VAR_INPUT
	sensorByte : UINT; // byte where the sensor is in 
	sensorBit : UINT;  // bit from the sensor
	sensorLocation : IOExpantionLocation_t; // location of the sensor
END_VAR

VAR
	_tmpStr: STRING;
END_VAR
CASE sensorLocation OF
	IOExpantionLocation_t.ROOT:
		IF sensorByte > 0 THEN
			extractSensorBit := FALSE; 
			_ErrorMessage.CreateEx(TC_EVENTS.ProgrammingErrors.invalidAccsessOfByte, 0 );
			_ErrorMessage.ipArguments.AddString(__POUNAME());
			_tmpStr := formatPosition(__POSITION());
			_ErrorMessage.ipArguments.AddString(_tmpStr);
			_ErrorMessage.Send(0);
			RETURN;
		END_IF

		(*
		The function convertByteBit(...) only accepts an BYTE not a UINT. A BYTE has 8 bits and a UINT has 16. We need to convert the UINT to a BYTE, 
		this is non trivial, beacuse if the sensorBit > 7 then we must accsess the other 8 bits.   
		
		 1111  1111   1111  1111 
 		|		   | |			|
		------------ ------------
		   8 - 15    	0 - 7
		   
		For that we must shift the value 8 bits to the right if sensorBit > 7. 
		For this we use this thing of a math expression: FLOOR(sensorBit / 8) * 8
		
		To ajust the offset for the function we use this math expression: sensorBit - FLOOR(sensorBit / 8) * 8 
		The rest is convertion of data types.
		
 		*)
		extractSensorBit := convertByteBit(	byteVal := TO_BYTE(SHR(_IOExpantionInBytes[sensorByte]^, TO_UINT(FLOOR(sensorBit / 8) * 8))), 
											offset := TO_UINT(sensorBit - FLOOR(sensorBit / 8) * 8 ));
		
	IOExpantionLocation_t.EXPANTION:
		IF sensorByte > 1 THEN 
			extractSensorBit := FALSE; 
			_ErrorMessage.CreateEx(TC_EVENTS.ProgrammingErrors.invalidAccsessOfByte, 0 );
			_ErrorMessage.ipArguments.AddString(__POUNAME());
			_tmpStr := formatPosition(__POSITION());
			_ErrorMessage.ipArguments.AddString(_tmpStr);
			_ErrorMessage.Send(0);
			RETURN;
		END_IF
	
		extractSensorBit := convertByteBit(byteVal := _IOExpantionExpantionInBytes[sensorByte]^, offset := sensorBit);
END_CASE

RETURN;
END_METHOD

//FB_Init ist immer implizit verfügbar und wird primär für die Initialisierung verwendet.
//Der Rückgabewert wird nicht ausgewertet. Für gezielte Einflussnahme können Sie
//die Methoden explizit deklarieren und darin mit dem Standard-Initialisierungscode 
//zusätzlichen Code bereitstellen. Sie können den Rückgabewert auswerten.
METHOD FB_Init: BOOL
VAR_INPUT    
bInitRetains: BOOL; // TRUE: Die Retain-Variablen werden initialisiert (Reset warm / Reset kalt)    
bInCopyCode: BOOL;  // TRUE: Die Instanz wird danach in den Kopiercode kopiert (Online-Change)
END_VAR
_readDiagMessageClock.durrationBetweenSignals_ms := 50;
END_METHOD

METHOD PRIVATE genMessageDescription : IOExpantionMessageDescriptor_t;
VAR_INPUT
	_data : POINTER TO ARRAY[0..236] OF BYTE; 
END_VAR
// extract diagCode
memcpy(destAddr := ADR(genMessageDescription.diagCode), srcAddr := _data, n := SIZEOF(genMessageDescription.diagCode));

// extract textID
MEMCPY(destAddr := ADR(genMessageDescription.textID), srcAddr := ADR(_data^[6]), n := SIZEOF(genMessageDescription.textID));
END_METHOD

METHOD getActor : BOOL
VAR_INPUT
	actorID : actorID_t;
END_VAR
CASE actorID OF
	actorID_t.ACTOR_0:
		getActor := convertByteBit(_FestoPneumaticOutBytes[0]^, 0);
		
	actorID_t.ACTOR_1:
		getActor := convertByteBit(_FestoPneumaticOutBytes[0]^, 2);
		
	actorID_t.ACTOR_2:
		getActor := convertByteBit(_FestoPneumaticOutBytes[0]^, 4);
		
	actorID_t.ACTOR_3:
		getActor := convertByteBit(_FestoPneumaticOutBytes[0]^, 6);
		
	actorID_t.ACTOR_GRIPPER_RIGHT_LEFT:
		getActor := convertByteBit(_FestoPneumaticOutBytes[1]^, 0);	
		
	actorID_t.ACTOR_GRIPPER_OPEN_CLOSE:
		getActor := convertByteBit(_FestoPneumaticOutBytes[1]^, 2);
		
	actorID_t.ACTOR_GRIPPER_UP_DOWN:
		getActor := convertByteBit(_FestoPneumaticOutBytes[1]^, 4);
		
	actorID_t.ACTOR_Y1_OUT:
		getActor := convertByteBit(_FestoPneumaticOutBytes[1]^, 6);
		
	actorID_t.ACTOR_Y2_OUT:
		getActor := convertByteBit(_FestoPneumaticOutBytes[2]^, 0);
		
	actorID_t.ACTOR_Y3_OUT:
		getActor := convertByteBit(_FestoPneumaticOutBytes[2]^, 2);
	
END_CASE
END_METHOD

METHOD PRIVATE getMessage : BOOL
VAR_INPUT
	index : BYTE;
END_VAR
VAR_OUTPUT
	readLength : UDINT;
	busy : BOOL;
END_VAR
VAR 
	calculatedIndex : BYTE := 0;
	_error : BOOL := FALSE;
	_errorID : UDINT := 0;
	_busy : BOOL := FALSE;
END_VAR
calculatedIndex := index + 6; // 6 is offset
busy := true;
_readDiagMessage(
	sNetId:= '5.85.199.196.4.1', 
	nSlaveAddr:=1001 , 
	nSubIndex:= calculatedIndex, 
	nIndex:= 16#10F3, 
	pDstBuf:= ADR(_returnDiagBuffer), 
	cbBufLen:= 237, 
	bExecute:=TRUE , 
	tTimeout:= T#5S, 
	bBusy=> _busy, 
	bError=> _error, 
	nErrId=> _errorID, 
	cbRead=>ReadLength);
	
IF _busy = FALSE AND _returnDiagBuffer[0] <> 16#00 THEN
	// to cycle object
	_readDiagMessage(
		sNetId:= '5.85.199.196.4.1', 
		nSlaveAddr:=1001 , 
		nSubIndex:= calculatedIndex, 
		nIndex:= 16#10F3, 
		pDstBuf:= ADR(_returnDiagBuffer), 
		cbBufLen:= 237, 
		bExecute:=FALSE , 
		tTimeout:= T#5S, 
		bBusy=> , 
		bError=> , 
		nErrId=> , 
		cbRead=>ReadLength);
		busy := FALSE;
END_IF
	
	getMessage := TRUE;
	RETURN;
END_METHOD

METHOD PRIVATE getNewestMessageIndex : BYTE
VAR_INPUT
END_VAR
VAR_OUTPUT 
	busy : BOOL := FALSE;
	ReadLength : UDINT := 0;
END_VAR
VAR 
	_error : BOOL := FALSE;
	_errorID : UDINT := 0;
END_VAR
_readDiagIndex(
	sNetId:= '5.85.199.196.4.1', 
	nSlaveAddr:=1001 , 
	nSubIndex:= 2, 
	nIndex:= 16#10F3, 
	pDstBuf:= ADR(_returnIndexBuff), 
	cbBufLen:= 40, 
	bExecute:=TRUE , 
	tTimeout:= T#5S, 
	bBusy=> busy, 
	bError=> _error, 
	nErrId=> _errorID, 
	cbRead=>ReadLength);
	
	IF busy = FALSE THEN
		
		getNewestMessageIndex := _returnIndexBuff[0];
		// to cycle object
		_readDiagIndex(
			sNetId:= '5.85.199.196.4.1', 
			nSlaveAddr:=1001 , 
			nSubIndex:= 2, 
			nIndex:= 16#10F3, 
			pDstBuf:= ADR(_returnIndexBuff), 
			cbBufLen:= 40, 
			bExecute:=FALSE , 
			tTimeout:= T#5S, 
			bBusy=> , 
			bError=> , 
			nErrId=> , 
			cbRead=>ReadLength);
	ELSE 
		getNewestMessageIndex := 16#00;
	END_IF
	RETURN;
END_METHOD

METHOD PRIVATE getNextMessageIndex : BYTE;
VAR_INPUT
	currentIndex : BYTE;
END_VAR

getNextMessageIndex := currentIndex + 1;

IF getNextMessageIndex = 16#00 THEN
	getNextMessageIndex := TO_BYTE(16#06);
END_IF

return;
END_METHOD

METHOD getSensorStatus : BOOL
VAR_INPUT
	sensorID : sensorID_t;
END_VAR
CASE sensorID OF
	sensorID_t.SENSOR_B8_CONVAYORBELT_METTAL_PRESENT:
		getSensorStatus := extractSensorBit(sensorLocation := IOExpantionLocation_t.EXPANTION, sensorByte := 0, sensorBit := 0); 
	sensorID_t.SENSOR_B5_STORAGE_ENTRANCE:
		getSensorStatus := extractSensorBit(sensorLocation := IOExpantionLocation_t.EXPANTION, sensorByte := 0, sensorBit := 1); 
		
	sensorID_t.SENSOR_B17_GRIPPER_RIGHT:
		getSensorStatus := extractSensorBit(sensorLocation := IOExpantionLocation_t.EXPANTION, sensorByte := 0, sensorBit := 2); 
	sensorID_t.SENSOR_B16_GRIPPER_LEFT:
		getSensorStatus := extractSensorBit(sensorLocation := IOExpantionLocation_t.EXPANTION, sensorByte := 0, sensorBit := 3); 
		
	sensorID_t.SENSOR_B3_Y3_DOWN:
		getSensorStatus := extractSensorBit(sensorLocation := IOExpantionLocation_t.EXPANTION, sensorByte := 0, sensorBit := 4); 
	sensorID_t.SENSOR_B4_Y3_UP:
		getSensorStatus := extractSensorBit(sensorLocation := IOExpantionLocation_t.EXPANTION, sensorByte := 0, sensorBit := 5); 
		
	sensorID_t.EXPANTION_SENSOR_Y4_UP:
		getSensorStatus := extractSensorBit(sensorLocation := IOExpantionLocation_t.EXPANTION, sensorByte := 0, sensorBit := 6); 
	sensorID_t.EXPANTION_SENSOR_B11_Y5_INSIDE:
		getSensorStatus := extractSensorBit(sensorLocation := IOExpantionLocation_t.EXPANTION, sensorByte := 0, sensorBit := 7); 
		
	sensorID_t.EXPANTION_SENSOR_B7_ENTRANCE_CONVAYORBELT:
		getSensorStatus := extractSensorBit(sensorLocation := IOExpantionLocation_t.EXPANTION, sensorByte := 1, sensorBit := 0); 
	sensorID_t.EXPANTION_SENSOR_B6_PART_SENSOR_METTAL_PRESENT:
		getSensorStatus := extractSensorBit(sensorLocation := IOExpantionLocation_t.EXPANTION, sensorByte := 1, sensorBit := 1); 
		
	sensorID_t.EXPANTION_SENSOR_B12_PART_TURNTABLE_PRESENT:
		getSensorStatus := extractSensorBit(sensorLocation := IOExpantionLocation_t.EXPANTION, sensorByte := 1, sensorBit := 2); 
	sensorID_t.EXPANTION_SENSOR_Y4_DOWN:
		getSensorStatus := extractSensorBit(sensorLocation := IOExpantionLocation_t.EXPANTION, sensorByte := 1, sensorBit := 3); 
		
	sensorID_t.EXPANTION_SENSOR_B10_Y5_OUT:
		getSensorStatus := extractSensorBit(sensorLocation := IOExpantionLocation_t.EXPANTION, sensorByte := 1, sensorBit := 4); 
	sensorID_t.EXPANTION_SENSOR_B18_SENSOR_Y4:
		getSensorStatus := extractSensorBit(sensorLocation := IOExpantionLocation_t.EXPANTION, sensorByte := 1, sensorBit := 5); 	
		
	sensorID_t.EXPANTION_SENSOR_B1_Y2_DOWN:
		getSensorStatus := extractSensorBit(sensorLocation := IOExpantionLocation_t.EXPANTION, sensorByte := 1, sensorBit := 6); 
	sensorID_t.EXPANTION_SENSOR_B2_Y2_UP:
		getSensorStatus := extractSensorBit(sensorLocation := IOExpantionLocation_t.EXPANTION, sensorByte := 1, sensorBit := 7); 
		
	sensorID_t.SENSOR_PNEUMATIC_PRESHURE_OK:
		getSensorStatus := extractSensorBit(sensorLocation := IOExpantionLocation_t.ROOT, sensorByte := 0, sensorBit := 12); 
	sensorID_t.SENSOR_B13_TURNTABLE_POS_REACHED:
		getSensorStatus := extractSensorBit(sensorLocation := IOExpantionLocation_t.ROOT, sensorByte := 0, sensorBit := 13); 
END_CASE

RETURN;
END_METHOD

METHOD PRIVATE isMesDesEqual : BOOL
VAR_INPUT
	messageDescription1 : IOExpantionMessageDescriptor_t;
	messageDescription2 : IOExpantionMessageDescriptor_t;
END_VAR
VAR
	i : UINT := 0;
END_VAR
isMesDesEqual := TRUE;
FOR i := 0 TO 3 DO
	isMesDesEqual := isMesDesEqual AND messageDescription1.diagCode[i] = messageDescription2.diagCode[i];
END_FOR

FOR i := 0 TO 1 DO
	isMesDesEqual := isMesDesEqual AND messageDescription1.textID[i] = messageDescription2.textID[i];
END_FOR

RETURN;
END_METHOD

METHOD PRIVATE isNewMessageAvalable : BOOL
VAR_INPUT
END_VAR
VAR_OUTPUT 
	busy : BOOL := FALSE;
	ReadLength : UDINT := 0;
END_VAR
VAR 
	_destBuff : BOOL := 0;
END_VAR
_readDiagMessage(
	sNetId:= '5.85.199.196.4.1', 
	nSlaveAddr:=1001 , 
	nSubIndex:= 16#04, 
	nIndex:= 16#10F3, 
	pDstBuf:= ADR(_destBuff), 
	cbBufLen:= 237, 
	bExecute:=TRUE , 
	tTimeout:= T#5S, 
	bBusy=> busy, 
	bError=> , 
	nErrId=> , 
	cbRead=>ReadLength);
	
	IF busy = FALSE THEN
		isNewMessageAvalable := _destBuff;
		// to cycle object
		_readDiagMessage(
			sNetId:= '5.85.199.196.4.1', 
			nSlaveAddr:=1001 , 
			nSubIndex:= 16#04, 
			nIndex:= 16#10F3, 
			pDstBuf:= ADR(_destBuff), 
			cbBufLen:= 237, 
			bExecute:=FALSE , 
			tTimeout:= T#5S, 
			bBusy=> busy, 
			bError=> , 
			nErrId=> , 
			cbRead=>);
	ELSE 
		isNewMessageAvalable := FALSE;
	END_IF
	RETURN;
END_METHOD

METHOD setActor : BOOL
VAR_INPUT
	actorID : actorID_t;
	value : BOOL;

END_VAR

CASE actorID OF
	actorID_t.ACTOR_0:
		setActorBit(_FestoPneumaticOutBytes[0], 0, value);
		
	actorID_t.ACTOR_1:
		setActorBit(_FestoPneumaticOutBytes[0], 2, value);
		
	actorID_t.ACTOR_2:
		setActorBit(_FestoPneumaticOutBytes[0], 4, value);
		
	actorID_t.ACTOR_3:
		setActorBit(_FestoPneumaticOutBytes[0], 6, value);
		
	actorID_t.ACTOR_GRIPPER_RIGHT_LEFT:
		setActorBit(_FestoPneumaticOutBytes[1], 0, value);	
		
	actorID_t.ACTOR_GRIPPER_OPEN_CLOSE:
		setActorBit(_FestoPneumaticOutBytes[1], 2, value);
		
	actorID_t.ACTOR_GRIPPER_UP_DOWN:
		setActorBit(_FestoPneumaticOutBytes[1], 4, value);
		
	actorID_t.ACTOR_Y1_OUT:
		setActorBit(_FestoPneumaticOutBytes[1], 6, value);
		
	actorID_t.ACTOR_Y2_OUT:
		setActorBit(_FestoPneumaticOutBytes[2], 0, value);
		
	actorID_t.ACTOR_Y3_OUT:
		setActorBit(_FestoPneumaticOutBytes[2], 2, value);
	
END_CASE
END_METHOD

METHOD PRIVATE setActorBit : BOOL
VAR_INPUT
	byteVal : POINTER TO BYTE;
	offset : UINT;
	value : BOOL;
END_VAR
VAR
	tmpByte : BYTE; 
	_tmpStr: STRING;
END_VAR

IF offset > 7 THEN 
	setActorBit := FALSE; 
	_ErrorMessage.CreateEx(TC_EVENTS.ProgrammingErrors.invalidAccsessOfByte, 0 );
	_ErrorMessage.ipArguments.AddString(__POUNAME());
	_tmpStr := formatPosition(__POSITION());
	_ErrorMessage.ipArguments.AddString(_tmpStr);
	_ErrorMessage.Send(0);
	RETURN;
END_IF

tmpByte := (NOT SHL(1, offset)) AND byteVal^;

byteVal^ := TO_BYTE(SHL(TO_INT(value), offset)) OR tmpByte;
END_METHOD

// subsctibes to a Message
METHOD subscribe : BOOL
VAR_INPUT
	callbackVariable : POINTER TO BOOL;
	diagCode : ARRAY [0..3] OF BYTE;
	textID : ARRAY [0..1] OF BYTE;
END_VAR
VAR 
	i : UINT := 0;
	spaceFound : BOOL := FALSE;
	_tmpStr: STRING;
END_VAR
IF callbackVariable = NULL THEN
	subscribe := FALSE;	
	RETURN; // nothing to call back to
END_IF

// search for avalable spot in list, may be expencive (worst case O(n))
FOR i := 0 TO 99 DO
	IF _subscriberArray[i].callbackVariable = NULL THEN
		spaceFound := TRUE;
		EXIT;
	END_IF
END_FOR

IF spaceFound = FALSE THEN
	subscribe := FALSE;
	_ErrorMessage.CreateEx(TC_EVENTS.ProgrammingErrors.subscriberArrayFull, 0 );
	_ErrorMessage.ipArguments.AddString(__POUNAME());
	_tmpStr := formatPosition(__POSITION());
	_ErrorMessage.ipArguments.AddString(_tmpStr);
	_ErrorMessage.ipArguments.AddUInt(SIZEOF(_subscriberArray) / SIZEOF(IOExpantionMessageSubData_t));
	_ErrorMessage.Send(0);
	RETURN;
END_IF


// insert value
_subscriberArray[i].callbackVariable := callbackVariable;
_subscriberArray[i].messageDescription.diagCode := diagCode;
_subscriberArray[i].messageDescription.textID := textID;

subscribe := TRUE;
RETURN;
END_METHOD

// unsubscribe from a message
METHOD unsubscribe : BOOL
VAR_INPUT
	callbackVariable : POINTER TO BOOL;
END_VAR
VAR 
	spaceFound : BOOL := FALSE;
	i : UINT := 0;
	_tmpStr : STRING;
END_VAR
IF callbackVariable = NULL THEN
	unsubscribe := FALSE;	
	RETURN; // nothing to call back to
END_IF

// search for avalable spot in list, may be expencive (worst case O(n))
FOR i := 0 TO 99 DO
	IF _subscriberArray[i].callbackVariable = callbackVariable THEN
		spaceFound := TRUE;
		EXIT;
	END_IF
END_FOR

IF spaceFound = FALSE THEN
	unsubscribe := FALSE;
	_ErrorMessage.CreateEx(TC_EVENTS.ProgrammingErrors.subscriberArrayFull, 0 );
	_ErrorMessage.ipArguments.AddString(__POUNAME());
	_tmpStr := formatPosition(__POSITION());
	_ErrorMessage.ipArguments.AddString(_tmpStr);
	_ErrorMessage.ipArguments.AddUInt(SIZEOF(_subscriberArray) / SIZEOF(IOExpantionMessageSubData_t));
	_ErrorMessage.Send(0);
	RETURN;
END_IF


// reset pointer 
_subscriberArray[i].callbackVariable := NULL;

unsubscribe := TRUE;
RETURN;
END_METHOD

END_FUNCTION_BLOCK

// ---- POUs/ErrorSystem/formatPosition.TcPOU
FUNCTION formatPosition : STRING
VAR_INPUT
	line : STRING; 
END_VAR
VAR
	_line : STRING;
	lineNumber : STRING;
	delimitorIndex : INT := 0;
END_VAR

// remove stuf indfront and in the back
_line := line;

_line := delete(_line, 6, 1);
_line := delete(_line, 7, len(_line)-6);

// extract line number
delimitorIndex := find(_line, ',');
lineNumber := left(_line, delimitorIndex - 1);
_line := delete(_line, delimitorIndex + 8, 1);

// formate string
formatPosition := CONCAT(lineNumber, concat(':', _line));
RETURN;

END_FUNCTION

// ---- POUs/MainStateMachine/mainStateMachine_t.TcPOU
// this class implements the main state machine, witch controls the olperations in automatic mode
FUNCTION_BLOCK mainStateMachine_t
VAR_INPUT
	IOExpantionHandler : POINTER TO IOExpantionHandler_t := NULL;
END_VAR
VAR_OUTPUT
END_VAR
VAR
	(* main envorment variables *)	

	isStateMachineOn : BOOL := FALSE; // is stae machine running or not
	stateMachineState : mainStateMachineStatus_t := mainStateMachineStatus_t.IDLE;
	
	startSceduled : BOOL := FALSE; // if true, the "api" has requested the start of the state machine
	stopSceduled : BOOL := FALSE; // if true, the "api" has requzested a stop of the state machine
	
	isStateMachinePaused : BOOL := FALSE;
	
	
	(* RotateTable variables *)	
	
	RotateTable_firstRun : BOOL := TRUE; 		// true when RotateTable is run the first time
	RotateTable_initialState : BOOL := FALSE;	// is the initial state of the TurnTable pos reached sensor
	RotateTable_waitOnRechingPos : TON;
	
	
	(* GripperDown variables *)

	GripperDown_waitUntilNextStep : TON;	
	
	
	(* GripperClose variables *)

	GripperClose_waitUntilNextStep : TON;	
	
	
	(* GripperUp variables *)

	GripperUp_waitUntilNextStep : TON;	
	
	(* GripperDownLeft variables *)

	GripperDownLeft_waitUntilNextStep : TON;	
	
	
	(* GripperOpen variables *)

	GripperOpen_waitUntilNextStep : TON;
	
	(* GripperUpLeft variables *)

	GripperUpLeft_waitUntilNextStep : TON;
	
	(* Y10Out variables *)

	Y10Out_waitUntilNextStep : TON;
	
	
	(* Y10Back variables *)

	Y10Back_waitUntilNextStep : TON;
END_VAR

METHOD PRIVATE convayorbeltStop : BOOL
VAR_INPUT
END_VAR
IOExpantionHandler^.setActor(actorID := actorID_t.ACTOR_Y2_OUT, false);
IOExpantionHandler^.setActor(actorID := actorID_t.ACTOR_Y3_OUT, false);
InputOutput.ConvaorbeltMotorRun := FALSE;

THIS^.stateMachineState := mainStateMachineStatus_t.IDLE; // move on to next step
END_METHOD

METHOD PRIVATE conveyorbeltStart : BOOL
VAR_INPUT
END_VAR
InputOutput.ConvaorbeltMotorRun := TRUE;

IF IOExpantionHandler^.getSensorStatus(sensorID := sensorID_t.EXPANTION_SENSOR_B7_ENTRANCE_CONVAYORBELT) = TRUE THEN
	THIS^.stateMachineState := mainStateMachineStatus_t.Y10_BACK; // move on to next step
END_IF
END_METHOD

METHOD getIsStateMachineON : BOOL
VAR_INPUT
END_VAR
getIsStateMachineON := THIS^.isStateMachineOn;

return;
END_METHOD

METHOD getStateMachineStatus : string
VAR_INPUT
END_VAR
getStateMachineStatus := to_string(THIS^.stateMachineState);

return;
END_METHOD

METHOD PRIVATE GripperClose : BOOL
VAR_INPUT
END_VAR
GripperClose_waitUntilNextStep.PT := T#500MS;

// reset TON
IF GripperClose_waitUntilNextStep.IN = TRUE AND GripperClose_waitUntilNextStep.Q = TRUE THEN
	GripperClose_waitUntilNextStep.IN := FALSE;
	GripperClose_waitUntilNextStep();
END_IF

GripperClose_waitUntilNextStep.IN := TRUE;
GripperClose_waitUntilNextStep();

IOExpantionHandler^.setActor(actorID := actorID_t.ACTOR_GRIPPER_OPEN_CLOSE, TRUE);

IF GripperClose_waitUntilNextStep.Q = TRUE THEN
	GripperClose_waitUntilNextStep.IN := FALSE;
	GripperClose_waitUntilNextStep();
	
	THIS^.stateMachineState := mainStateMachineStatus_t.GRIPPER_UP; // move on to next step
END_IF
END_METHOD

METHOD PRIVATE GripperDown : BOOL
VAR_INPUT
END_VAR
IF GripperDown_waitUntilNextStep.IN = TRUE AND GripperDown_waitUntilNextStep.Q = TRUE THEN
	GripperDown_waitUntilNextStep.IN := FALSE;
	GripperDown_waitUntilNextStep();
END_IF

THIS^.IOExpantionHandler^.setActor(actorID_t.ACTOR_GRIPPER_RIGHT_LEFT, FALSE);

IF IOExpantionHandler^.getSensorStatus(sensorID := sensorID_t.SENSOR_B17_GRIPPER_RIGHT) = FALSE THEN
	// wait (gripper is not on the right)
	RETURN;
END_IF

// configure GripperDown_waitUntilNextStep
GripperDown_waitUntilNextStep.PT := T#500ms;

GripperDown_waitUntilNextStep.IN := TRUE;
GripperDown_waitUntilNextStep();


IOExpantionHandler^.setActor(actorID := actorID_t.ACTOR_GRIPPER_UP_DOWN, TRUE);

IF GripperDown_waitUntilNextStep.Q = FALSE THEN
	RETURN;
END_IF

GripperDown_waitUntilNextStep.IN := FALSE;
GripperDown_waitUntilNextStep();

THIS^.stateMachineState := mainStateMachineStatus_t.GRIPPER_CLOSE; // move on to next step
END_METHOD

METHOD PRIVATE GripperDownLeft : BOOL
VAR_INPUT
END_VAR
GripperDownLeft_waitUntilNextStep.PT := T#1S;

IF GripperDownLeft_waitUntilNextStep.IN = TRUE AND GripperDownLeft_waitUntilNextStep.Q = TRUE THEN
	GripperDownLeft_waitUntilNextStep.IN := FALSE;
	GripperDownLeft_waitUntilNextStep();
END_IF

GripperDownLeft_waitUntilNextStep.IN := TRUE;
GripperDownLeft_waitUntilNextStep();

IOExpantionHandler^.setActor(actorID := actorID_t.ACTOR_GRIPPER_UP_DOWN, TRUE);

IF GripperDownLeft_waitUntilNextStep.Q = TRUE THEN
	GripperDownLeft_waitUntilNextStep.IN := FALSE;
	GripperDownLeft_waitUntilNextStep();	
	
	THIS^.stateMachineState := mainStateMachineStatus_t.GRIPPER_OPEN; // move on to next step
END_IF
END_METHOD

METHOD PRIVATE GripperLeft : BOOL
VAR_INPUT
END_VAR

IOExpantionHandler^.setActor(actorID := actorID_t.ACTOR_GRIPPER_RIGHT_LEFT, true);

IF IOExpantionHandler^.getSensorStatus(sensorID := sensorID_t.SENSOR_B16_GRIPPER_LEFT) = TRUE THEN
	THIS^.stateMachineState := mainStateMachineStatus_t.GRIPPER_DOWN_LEFT; // move on to next step
END_IF
END_METHOD

METHOD PRIVATE GripperOpen : BOOL
VAR_INPUT
END_VAR
GripperOpen_waitUntilNextStep.PT := T#200MS;

IF GripperOpen_waitUntilNextStep.IN = TRUE AND GripperOpen_waitUntilNextStep.Q = TRUE THEN
	GripperOpen_waitUntilNextStep.IN := FALSE;
	GripperOpen_waitUntilNextStep();
END_IF

GripperOpen_waitUntilNextStep.IN := TRUE;
GripperOpen_waitUntilNextStep();

IOExpantionHandler^.setActor(actorID := actorID_t.ACTOR_GRIPPER_OPEN_CLOSE, FALSE);

IF GripperOpen_waitUntilNextStep.Q = TRUE THEN
	GripperOpen_waitUntilNextStep.IN := FALSE;
	GripperOpen_waitUntilNextStep();

	THIS^.stateMachineState := mainStateMachineStatus_t.GRIPPER_UP_LEFT; // move on to next step
END_IF
END_METHOD

METHOD PRIVATE GripperRight : BOOL
VAR_INPUT
END_VAR
END_METHOD

METHOD PRIVATE GripperUp : BOOL
VAR_INPUT
END_VAR
VAR 
	
END_VAR
GripperUp_waitUntilNextStep.PT := T#500MS;

IF GripperUp_waitUntilNextStep.IN = TRUE AND GripperUp_waitUntilNextStep.Q = TRUE THEN
	GripperUp_waitUntilNextStep.IN := FALSE;
	GripperUp_waitUntilNextStep();
END_IF

GripperUp_waitUntilNextStep.IN := TRUE;
GripperUp_waitUntilNextStep();

IOExpantionHandler^.setActor(actorID := actorID_t.ACTOR_GRIPPER_UP_DOWN, FALSE);

IF GripperUp_waitUntilNextStep.Q = TRUE THEN
	THIS^.stateMachineState := mainStateMachineStatus_t.GRIPPER_LEFT; // move on to next step
END_IF
END_METHOD

METHOD PRIVATE GripperUpLeft : BOOL
VAR_INPUT
END_VAR
GripperUpLeft_waitUntilNextStep.PT := T#500MS;

IF GripperUpLeft_waitUntilNextStep.IN = TRUE AND GripperUpLeft_waitUntilNextStep.Q = TRUE THEN
	GripperUpLeft_waitUntilNextStep.IN := FALSE;
	GripperUpLeft_waitUntilNextStep();
END_IF


IOExpantionHandler^.setActor(actorID := actorID_t.ACTOR_GRIPPER_UP_DOWN, FALSE);

GripperUpLeft_waitUntilNextStep.IN := TRUE;
GripperUpLeft_waitUntilNextStep();	

IF GripperUpLeft_waitUntilNextStep.Q = TRUE THEN
	GripperUpLeft_waitUntilNextStep.IN := FALSE;
	GripperUpLeft_waitUntilNextStep();	

	IF IOExpantionHandler^.getSensorStatus(sensorID := sensorID_t.EXPANTION_SENSOR_B7_ENTRANCE_CONVAYORBELT) = TRUE THEN
		THIS^.stateMachineState := mainStateMachineStatus_t.CONVAYORBELT_START; // move on to next step
	ELSE 
		THIS^.stateMachineState := mainStateMachineStatus_t.Y10_OUT; // move on to next step
	END_IF;
END_IF
END_METHOD

// if this function is called, the statemachine pauses its execution and stores its state, all movement will be paused or will wait until all movment is paused. A mutch "safer" alternative to reset()
METHOD pause : BOOL
VAR_INPUT
	isPaused : BOOL := TRUE;	
END_VAR
IF THIS^.isStateMachineOn = FALSE THEN
	pause := FALSE;
	RETURN;
END_IF

THIS^.isStateMachinePaused := TRUE; 
pause := TRUE;
return;
END_METHOD

// WARNING: this function is dangerous, if called the state machine imediatly stopps its execution and all values are reset. No safety is garantied, the stateMachine forces itself ot its original state.
METHOD reset : BOOL
VAR_INPUT
END_VAR
{warning: 'implement reset of mainStateMachine'}

stateMachineState := mainStateMachineStatus_t.IDLE;

InputOutput.TurnTableMotorTurn := FALSE;
IOExpantionHandler^.setActor(actorID := actorID_t.ACTOR_GRIPPER_UP_DOWN, FALSE);
IOExpantionHandler^.setActor(actorID := actorID_t.ACTOR_GRIPPER_RIGHT_LEFT, TRUE);
IOExpantionHandler^.setActor(actorID := actorID_t.ACTOR_GRIPPER_OPEN_CLOSE, FALSE);
IOExpantionHandler^.setActor(actorID := actorID_t.ACTOR_Y1_OUT, FALSE);
IOExpantionHandler^.setActor(actorID := actorID_t.ACTOR_Y3_OUT, FALSE);
IOExpantionHandler^.setActor(actorID := actorID_t.ACTOR_Y2_OUT, FALSE);
InputOutput.ConvaorbeltMotorRun := false;


THIS^.isStateMachineOn := false;

reset := false;
RETURN;
END_METHOD

METHOD PRIVATE RotateTable : BOOL
VAR_INPUT
END_VAR
// configure RotateTable_waitOnRechingPos
RotateTable_waitOnRechingPos.PT := T#500MS;


RotateTable_waitOnRechingPos();

// move the gripper away, because he is too low (the sensor for detecting workpices will detect the gripper :( )
IOExpantionHandler^.setActor(actorID_t.ACTOR_GRIPPER_RIGHT_LEFT, TRUE);

// wait until the gripper has moved away
IF IOExpantionHandler^.getSensorStatus(sensorID := sensorID_t.SENSOR_B16_GRIPPER_LEFT) = FALSE THEN
	RETURN;
END_IF

// run initialsie code if it is the first time it is ran
IF THIS^.RotateTable_firstRun = TRUE THEN
	THIS^.RotateTable_firstRun := FALSE;
	THIS^.RotateTable_initialState := IOExpantionHandler^.getSensorStatus(sensorID := sensorID_t.SENSOR_B13_TURNTABLE_POS_REACHED);
	RotateTable_waitOnRechingPos.IN := FALSE; // make shure this is false when starting
END_IF


IF RotateTable_waitOnRechingPos.IN = FALSE THEN
	// rotate motor
	InputOutput.TurnTableMotorTurn := TRUE;
END_IF


IF THIS^.RotateTable_initialState = TRUE THEN
	IF IOExpantionHandler^.getSensorStatus(sensorID := sensorID_t.SENSOR_B13_TURNTABLE_POS_REACHED) = TRUE THEN 
		RETURN; // return if the SENSOR_B13_TURNTABLE_POS_REACHED isn't false and was truie when the state started
	ELSE 
		RotateTable_initialState := FALSE; // job of initialstate achived (set to false to stop further involvment)
	END_IF 
END_IF

// check for position of motor
IF IOExpantionHandler^.getSensorStatus(sensorID := sensorID_t.SENSOR_B13_TURNTABLE_POS_REACHED) = TRUE THEN
	RotateTable_waitOnRechingPos.IN := TRUE;
	InputOutput.TurnTableMotorTurn := FALSE; 
	IF RotateTable_waitOnRechingPos.Q = FALSE THEN
		RETURN; // return if time hasn't passed
	END_IF

	// position reached (check if a part is at position)
	IF IOExpantionHandler^.getSensorStatus(sensorID := sensorID_t.EXPANTION_SENSOR_B12_PART_TURNTABLE_PRESENT) = TRUE THEN
		InputOutput.TurnTableMotorTurn := FALSE;
		THIS^.RotateTable_firstRun := TRUE;
		RotateTable_waitOnRechingPos.IN := FALSE;
		RotateTable_waitOnRechingPos();
		THIS^.stateMachineState := mainStateMachineStatus_t.GRIPPER_DOWN; // move on to next step
	ELSE 
		
		// reset function and move on to the next position
		RotateTable_waitOnRechingPos.IN := FALSE;
		RotateTable_waitOnRechingPos();
		THIS^.RotateTable_firstRun := TRUE;
		InputOutput.TurnTableMotorTurn := FALSE;
		THIS^.stateMachineState := mainStateMachineStatus_t.IDLE; // move on to next step
	END_IF
END_IF
END_METHOD

// scedules the staret of the state machine
METHOD startStateMachine : BOOL
VAR_INPUT
END_VAR
IF THIS^.isStateMachineOn = TRUE THEN
	startStateMachine := FALSE;
	RETURN;
END_IF

startSceduled := TRUE;

startStateMachine := TRUE;
RETURN;
END_METHOD

METHOD stopStateMachine : BOOL
VAR_INPUT
END_VAR
IF THIS^.isStateMachineOn = FALSE THEN
	stopStateMachine := FALSE;
	RETURN;
END_IF

stopSceduled := TRUE;
stopStateMachine := TRUE;
return;
END_METHOD

// main update function call this every cycle
METHOD update : BOOL
VAR_INPUT
END_VAR
{warning: implement update FUNCTION}

IF THIS^.IOExpantionHandler = NULL THEN
	update := FALSE;
	RETURN;
END_IF

CASE THIS^.stateMachineState OF
	mainStateMachineStatus_t.IDLE: 
		IF THIS^.startSceduled = TRUE THEN // start state machine
			THIS^.startSceduled := FALSE;
			THIS^.isStateMachineOn := TRUE;
			stateMachineState := mainStateMachineStatus_t.ROTATE_TABLE; 
		END_IF
		THIS^.startSceduled := FALSE;
		
		IF THIS^.stopSceduled = TRUE THEN
			THIS^.stopSceduled := FALSE;
			THIS^.isStateMachineOn := FALSE;
		END_IF
		
		IF THIS^.isStateMachineOn = TRUE THEN
			stateMachineState := mainStateMachineStatus_t.ROTATE_TABLE; 
		END_IF
		
	mainStateMachineStatus_t.CONVAYORBELT_START: 
		THIS^.conveyorbeltStart();
		
	mainStateMachineStatus_t.CONVEYORBELT_STOP: 
		THIS^.convayorbeltStop();
		
	mainStateMachineStatus_t.GRIPPER_CLOSE: 
		THIS^.GripperClose();
		
	mainStateMachineStatus_t.GRIPPER_DOWN: 
		THIS^.GripperDown();
	
	mainStateMachineStatus_t.GRIPPER_DOWN_LEFT: 
		THIS^.GripperDownLeft();
	
	mainStateMachineStatus_t.GRIPPER_LEFT: 
		THIS^.GripperLeft();
	
	mainStateMachineStatus_t.GRIPPER_OPEN: 
		THIS^.GripperOpen();
	
	mainStateMachineStatus_t.GRIPPER_RIGHT: 
		THIS^.GripperRight();
	
	mainStateMachineStatus_t.GRIPPER_UP: 
		THIS^.GripperUp();
	
	mainStateMachineStatus_t.GRIPPER_UP_LEFT: 
		THIS^.GripperUpLeft();
	
	mainStateMachineStatus_t.ROTATE_TABLE: 
		THIS^.startSceduled := FALSE; // HACK: don't know why in idle the state doesn't get reset, and I don't care, this thing works :)
		THIS^.RotateTable();
	
	mainStateMachineStatus_t.Y10_BACK: 
		THIS^.Y10Back();
	
	mainStateMachineStatus_t.Y10_OUT: 
		THIS^.Y10Out();
	
	mainStateMachineStatus_t.Y2_OUT: 
		THIS^.Y2Out();
	
	mainStateMachineStatus_t.Y3_OUT: 
		THIS^.Y3Out();
	
END_CASE
END_METHOD

METHOD Y10Back : BOOL
VAR_INPUT
END_VAR
VAR
	B8 : BOOL := FALSE;
	B5 : BOOL := FALSE;
	B6 : bool := false;
END_VAR
IOExpantionHandler^.setActor(actorID := actorID_t.ACTOR_Y1_OUT, FALSE);

B8 := IOExpantionHandler^.getSensorStatus(sensorID := sensorID_t.SENSOR_B8_CONVAYORBELT_METTAL_PRESENT);
B5 := IOExpantionHandler^.getSensorStatus(sensorID := sensorID_t.SENSOR_B5_STORAGE_ENTRANCE);
B6 := IOExpantionHandler^.getSensorStatus(sensorID := sensorID_t.EXPANTION_SENSOR_B6_PART_SENSOR_METTAL_PRESENT);

Y10Back_waitUntilNextStep.PT := T#10S;

IF Y10Back_waitUntilNextStep.IN = TRUE AND Y10Back_waitUntilNextStep.Q = TRUE THEN
	Y10Back_waitUntilNextStep.IN := FALSE;
	Y10Back_waitUntilNextStep();
END_IF

Y10Back_waitUntilNextStep.IN := TRUE;
Y10Back_waitUntilNextStep();

IF B8 = FALSE AND B5 = FALSE AND B6 = TRUE THEN
	THIS^.stateMachineState := mainStateMachineStatus_t.Y2_OUT; // move on to next step
	Y10Back_waitUntilNextStep.IN := FALSE;
	Y10Back_waitUntilNextStep();
	
ELSIF B8 = TRUE AND B5 = FALSE and B6 = true THEN
	THIS^.stateMachineState := mainStateMachineStatus_t.Y3_OUT; // move on to next step
	Y10Back_waitUntilNextStep.IN := FALSE;
	Y10Back_waitUntilNextStep();
	
ELSIF Y10Back_waitUntilNextStep.Q = TRUE AND B5 = TRUE THEN
	THIS^.stateMachineState := mainStateMachineStatus_t.CONVEYORBELT_STOP; // move on to next step
	Y10Back_waitUntilNextStep.IN := FALSE;
	Y10Back_waitUntilNextStep();
END_IF
END_METHOD

METHOD PRIVATE Y10Out : BOOL
VAR_INPUT
END_VAR
Y10Out_waitUntilNextStep.PT := T#100MS;

IF Y10Out_waitUntilNextStep.IN = TRUE AND Y10Out_waitUntilNextStep.Q = TRUE THEN
	Y10Out_waitUntilNextStep.IN := FALSE;
	Y10Out_waitUntilNextStep();
END_IF

IOExpantionHandler^.setActor(actorID := actorID_t.ACTOR_Y1_OUT, TRUE);

Y10Out_waitUntilNextStep.IN := TRUE;
Y10Out_waitUntilNextStep();

IF Y10Out_waitUntilNextStep.Q = TRUE THEN
	Y10Out_waitUntilNextStep.IN := FALSE;
	Y10Out_waitUntilNextStep();
	
	THIS^.stateMachineState := mainStateMachineStatus_t.CONVAYORBELT_START; // move on to next step
END_IF
END_METHOD

METHOD PRIVATE Y2Out : BOOL
VAR_INPUT
END_VAR
IOExpantionHandler^.setActor(actorID := actorID_t.ACTOR_Y2_OUT, TRUE);

IF IOExpantionHandler^.getSensorStatus(sensorID := sensorID_t.SENSOR_B5_STORAGE_ENTRANCE) = TRUE THEN
	THIS^.stateMachineState := mainStateMachineStatus_t.CONVEYORBELT_STOP; // move on to next step
END_IF
END_METHOD

METHOD PRIVATE Y3Out : BOOL
VAR_INPUT
END_VAR
IOExpantionHandler^.setActor(actorID := actorID_t.ACTOR_Y3_OUT, TRUE);

IF IOExpantionHandler^.getSensorStatus(sensorID := sensorID_t.SENSOR_B5_STORAGE_ENTRANCE) = TRUE THEN
	THIS^.stateMachineState := mainStateMachineStatus_t.CONVEYORBELT_STOP; // move on to next step
END_IF
END_METHOD

END_FUNCTION_BLOCK

// ---- POUs/ARUIHandler/ARUIHandler_t.TcPOU
// this class implements variaus UI elements for the ARDevice
FUNCTION_BLOCK ARUIHandler_t
VAR_INPUT
	ARDevice : POINTER TO ARDeviceAPI_t := NULL;	
	systemStatus : POINTER TO systemStatus_t;
	IOExpantionHandler : POINTER TO IOExpantionHandler_t;
END_VAR
VAR_OUTPUT
END_VAR
VAR
	_PLCStatusDisplayErrorBlinker : FB_BA_Blink;
END_VAR

METHOD PRIVATE ControlpannelMessages : BOOL
VAR_INPUT
END_VAR

// set controlpannel message relese EM-Stop
IF NOT inputOutput.EmStop THEN
	THIS^.ARDevice^.displayEMStop := TRUE;
ELSE
	THIS^.ARDevice^.displayEMStop := FALSE;
END_IF


// set controlpannel message press Quitierung
IF InputOutput.QuittierenLamp = TRUE THEN
	THIS^.ARDevice^.displayQuittierung := TRUE;
ELSE
	THIS^.ARDevice^.displayQuittierung := FALSE;
END_IF
END_METHOD

METHOD PRIVATE ErrorSystemValues : BOOL
VAR_INPUT
END_VAR
THIS^.ARDevice^.errorHide_ERR_PNEU_LOW_PR_402 := NOT ErrorSystemStatusVar.errorHide_ERR_PNEU_LOW_PR_402;
THIS^.ARDevice^.errorHide_ERR_LD_START_LEFT_408_TIMEOUT := NOT ErrorSystemStatusVar.errorHide_ERR_LD_START_LEFT_408_TIMEOUT;
THIS^.ARDevice^.errorHide_ERR_LD_START_RIGHT_408_TIMEOUT := NOT ErrorSystemStatusVar.errorHide_ERR_LD_START_RIGHT_408_TIMEOUT;
THIS^.ARDevice^.errorHide_ERR_LD_MOVE_408_TIMEOUT := NOT ErrorSystemStatusVar.errorHide_ERR_LD_MOVE_408_TIMEOUT;
THIS^.ARDevice^.errorHide_ERR_RT_MOVE_408_TIMEOUT := NOT ErrorSystemStatusVar.errorHide_ERR_RT_MOVE_408_TIMEOUT;
THIS^.ARDevice^.errorHide_ERR_Y2_MOVE_408_TIMEOUT := NOT ErrorSystemStatusVar.errorHide_ERR_Y2_MOVE_408_TIMEOUT;
THIS^.ARDevice^.errorHide_ERR_Y2_START_DOWN_408_TIMEOUT := NOT ErrorSystemStatusVar.errorHide_ERR_Y2_START_DOWN_408_TIMEOUT;
THIS^.ARDevice^.errorHide_ERR_Y2_START_UP_408_TIMEOUT := NOT ErrorSystemStatusVar.errorHide_ERR_Y2_START_UP_408_TIMEOUT;
THIS^.ARDevice^.errorHide_ERR_Y3_MOVE_408_TIMEOUT := NOT ErrorSystemStatusVar.errorHide_ERR_Y3_MOVE_408_TIMEOUT;
THIS^.ARDevice^.errorHide_ERR_Y3_START_DOWN_408_TIMEOUT := NOT ErrorSystemStatusVar.errorHide_ERR_Y3_START_DOWN_408_TIMEOUT;
THIS^.ARDevice^.errorHide_ERR_Y3_START_UP_408_TIMEOUT := NOT ErrorSystemStatusVar.errorHide_ERR_Y3_START_UP_408_TIMEOUT;

ErrorSystemValues := TRUE;
RETURN;
END_METHOD

// displays in a status witch 
METHOD PRIVATE PLCStatusDisplay : BOOL
VAR_INPUT
END_VAR
_PLCStatusDisplayErrorBlinker.bEn := TRUE;
_PLCStatusDisplayErrorBlinker.udiTiOff := 500; // 500 ms
_PLCStatusDisplayErrorBlinker.udiTiOn := 500;  // 500 ms
_PLCStatusDisplayErrorBlinker();


CASE systemStatus^ OF
	systemStatus_t.RUNNING:
		THIS^.ARDevice^.lmpRunning := TRUE;
		THIS^.ARDevice^.lmpStopped := FALSE;
		THIS^.ARDevice^.lmpError := FALSE;
		
	systemStatus_t.STOPPED:
		THIS^.ARDevice^.lmpRunning := FALSE;
		THIS^.ARDevice^.lmpStopped := TRUE;
		THIS^.ARDevice^.lmpError := FALSE;

	systemStatus_t.ERROR:	
		THIS^.ARDevice^.lmpRunning := FALSE;
		THIS^.ARDevice^.lmpStopped := FALSE;
		THIS^.ARDevice^.lmpError := _PLCStatusDisplayErrorBlinker.bQ;

END_CASE
END_METHOD

METHOD PRIVATE sensorValues : BOOL
VAR_INPUT
END_VAR
THIS^.ARDevice^.PneumaticOkB20_sensorStatus := IOExpantionHandler^.getSensorStatus(sensorID := sensorID_t.SENSOR_PNEUMATIC_PRESHURE_OK);
THIS^.ARDevice^.PartTurntablePresentB12_sensorStatus := IOExpantionHandler^.getSensorStatus(sensorID := sensorID_t.EXPANTION_SENSOR_B12_PART_TURNTABLE_PRESENT);
THIS^.ARDevice^.LinearActuatorLeftB16_sensorStatus := IOExpantionHandler^.getSensorStatus(sensorID := sensorID_t.SENSOR_B16_GRIPPER_LEFT);
THIS^.ARDevice^.LinearActuatorRightB17_sensorStatus := IOExpantionHandler^.getSensorStatus(sensorID := sensorID_t.SENSOR_B17_GRIPPER_RIGHT);
THIS^.ARDevice^.TurntablePositionReachedB13_sensorStatus := IOExpantionHandler^.getSensorStatus(sensorID := sensorID_t.SENSOR_B13_TURNTABLE_POS_REACHED);
THIS^.ARDevice^.StorageEntranceB5_sensorStatus := IOExpantionHandler^.getSensorStatus(sensorID := sensorID_t.SENSOR_B5_STORAGE_ENTRANCE);
THIS^.ARDevice^.ConveyorBeltMetalPresentB8_sensorStatus := IOExpantionHandler^.getSensorStatus(sensorID := sensorID_t.SENSOR_B8_CONVAYORBELT_METTAL_PRESENT);
THIS^.ARDevice^.EntranceConveyorBeltB7_sensorStatus := IOExpantionHandler^.getSensorStatus(sensorID := sensorID_t.EXPANTION_SENSOR_B7_ENTRANCE_CONVAYORBELT);
THIS^.ARDevice^.SensorPartMetalPresentB6_sensorStatus := IOExpantionHandler^.getSensorStatus(sensorID := sensorID_t.EXPANTION_SENSOR_B6_PART_SENSOR_METTAL_PRESENT);
END_METHOD

// update function, call this every cycle
METHOD update : BOOL
VAR_INPUT
END_VAR
IF THIS^.ARDevice = NULL THEN
	update := FALSE;
	RETURN;
END_IF

THIS^.PLCStatusDisplay();
THIS^.ControlpannelMessages();
THIS^.sensorValues();
THIS^.ErrorSystemValues();

update := TRUE;
RETURN;
END_METHOD

END_FUNCTION_BLOCK

// ---- POUs/HMIHandler/HMIHandler_t.TcPOU
FUNCTION_BLOCK HMIHandler_t
VAR_INPUT
	systemStatus : POINTER TO systemStatus_t;
END_VAR
VAR_OUTPUT
END_VAR
VAR
	_PLCStatusDisplayErrorBlinker : FB_BA_Blink;
END_VAR

METHOD PRIVATE statusDisplayMachine : BOOL
VAR_INPUT
END_VAR
_PLCStatusDisplayErrorBlinker.bEn := TRUE;
_PLCStatusDisplayErrorBlinker.udiTiOff := 500; // 500 ms
_PLCStatusDisplayErrorBlinker.udiTiOn := 500;  // 500 ms
_PLCStatusDisplayErrorBlinker();


CASE systemStatus^ OF
	systemStatus_t.RUNNING:
		HMIInterface.HMIStartStatusLamp := TRUE;
		HMIInterface.HMIStopStatusLamp := FALSE;
		HMIInterface.HMIErrorStatusLamp := FALSE;
		
	systemStatus_t.STOPPED:
		HMIInterface.HMIStartStatusLamp := FALSE;
		HMIInterface.HMIStopStatusLamp := TRUE;
		HMIInterface.HMIErrorStatusLamp := FALSE;

	systemStatus_t.ERROR:	
		HMIInterface.HMIStartStatusLamp := FALSE;
		HMIInterface.HMIStopStatusLamp := FALSE;
		HMIInterface.HMIErrorStatusLamp := _PLCStatusDisplayErrorBlinker.bQ;

END_CASE
END_METHOD

// call this methode every cycle
METHOD update : BOOL
VAR_INPUT
END_VAR
this^.statusDisplayMachine();
END_METHOD

END_FUNCTION_BLOCK

// ---- POUs/ErrorSystem/ErrorManager_t.TcPOU
// This class is for managing all error detecting systems and is regestring errors in diffrent error classes
FUNCTION_BLOCK ErrorManager_t
VAR_INPUT
END_VAR
VAR_OUTPUT
END_VAR
VAR
	_actorMovingTimeoutManager : ActorMovingTimeoutManager_t;
	_actorStartMovingTimeoutManager : ActorStartMovingTimeoutManager_t;
	_primitiveWatchdogManager : PrimitiveWatchdogManager_t;
	_IOExpantionMessageErrorHandler : IOExpantionMessageErrorHandler_t;
	_IOExpantionHandler : POINTER TO IOExpantionHandler_t;
	
	_trowErrors : BOOL := FALSE; // if true, errors are checked
	_hasError : BOOL := FALSE; // if true, a error has been reported
	_errorsInitialised : BOOL := FALSE; // if true, errors have been initialised
	
END_VAR

METHOD confirmAll : BOOL
VAR_INPUT
END_VAR
_actorMovingTimeoutManager.confirmAll();
_actorStartMovingTimeoutManager.confirmAll();
_primitiveWatchdogManager.confirmAll();
_IOExpantionMessageErrorHandler.confirmAll();

confirmAll := TRUE;
return;
END_METHOD

//FB_Init ist immer implizit verfügbar und wird primär für die Initialisierung verwendet.
//Der Rückgabewert wird nicht ausgewertet. Für gezielte Einflussnahme können Sie
//die Methoden explizit deklarieren und darin mit dem Standard-Initialisierungscode 
//zusätzlichen Code bereitstellen. Sie können den Rückgabewert auswerten.
METHOD FB_Init: BOOL
VAR_INPUT    
bInitRetains: BOOL; // TRUE: Die Retain-Variablen werden initialisiert (Reset warm / Reset kalt)    
bInCopyCode: BOOL;  // TRUE: Die Instanz wird danach in den Kopiercode kopiert (Online-Change)
END_VAR
//
END_METHOD

// if the function returns true, an error has been reported
METHOD hasError : BOOL
VAR_INPUT
END_VAR
hasError := hasError OR THIS^._actorMovingTimeoutManager.hasError();
hasError := hasError OR THIS^._actorStartMovingTimeoutManager.hasError();
hasError := hasError OR THIS^._primitiveWatchdogManager.hasError();
hasError := hasError OR THIS^._actorMovingTimeoutManager.hasError();

_hasError := hasError;
return;
END_METHOD

METHOD PRIVATE initErrors : BOOL
VAR_INPUT
END_VAR
VAR CONSTANT
 	diagCodeErrorTestMessage : ARRAY[0..3] OF BYTE := [16#03, 16#E0, 16#08, 16#00];
	textIDErrorTestMessage : ARRAY[0..1] OF BYTE := [16#38, 16#00];
	diagCodeClearTestMessage : ARRAY[0..3] OF BYTE := [16#03, 16#E0, 16#08, 16#00];
	textIDClearTestMessage : ARRAY[0..1] OF BYTE := [16#38, 16#10];
END_VAR
// register all errors
_actorMovingTimeoutManager.register(stEventEntity := TC_EVENTS.OperationalErrors2.LinearDriveMoveTimedout, timerTime := T#10S, conformation := TRUE, sensorID1 := sensorID_t.SENSOR_B17_GRIPPER_RIGHT, sensorID2 := sensorID_t.SENSOR_B16_GRIPPER_LEFT, waitHWConformation := FALSE);
_actorMovingTimeoutManager.register(stEventEntity := TC_EVENTS.OperationalErrors2.RotaryTableMoveTimeout, timerTime := T#5S, conformation := TRUE, sensorID1 := sensorID_t.SENSOR_B13_TURNTABLE_POS_REACHED, waitHWConformation := FALSE);
_actorMovingTimeoutManager.register(stEventEntity := TC_EVENTS.OperationalErrors2.Y2moveTimeout, timerTime := T#2S, conformation := TRUE, sensorID1 := sensorID_t.EXPANTION_SENSOR_B1_Y2_DOWN, sensorID2 := sensorID_t.EXPANTION_SENSOR_B2_Y2_UP, waitHWConformation := FALSE);
_actorMovingTimeoutManager.register(stEventEntity := TC_EVENTS.OperationalErrors2.Y3moveTimeout, timerTime := T#2S, conformation := TRUE, sensorID1 := sensorID_t.SENSOR_B3_Y3_DOWN, sensorID2 := sensorID_t.SENSOR_B4_Y3_UP, waitHWConformation := FALSE);


_actorStartMovingTimeoutManager.register(stEventEntity := TC_EVENTS.OperationalErrors2.LinearDriveStartMoveLeftTimeout, timerTime := T#5S, conformation := TRUE, sensorID := sensorID_t.SENSOR_B16_GRIPPER_LEFT, actorID := actorID_t.ACTOR_GRIPPER_RIGHT_LEFT, expectedActorValue := TRUE, waitHWConformation := FALSE);
_actorStartMovingTimeoutManager.register(stEventEntity := TC_EVENTS.OperationalErrors2.LinearDriveStartMoveRightTimeout, timerTime := T#5S, conformation := TRUE, sensorID := sensorID_t.SENSOR_B17_GRIPPER_RIGHT, actorID := actorID_t.ACTOR_GRIPPER_RIGHT_LEFT, expectedActorValue := FALSE, waitHWConformation := FALSE);
_actorStartMovingTimeoutManager.register(stEventEntity := TC_EVENTS.OperationalErrors2.Y2StartMoveDownTimeout, timerTime := T#1S, conformation := TRUE, sensorID := sensorID_t.EXPANTION_SENSOR_B1_Y2_DOWN, actorID := actorID_t.ACTOR_Y2_OUT, expectedActorValue := FALSE, waitHWConformation := FALSE);
_actorStartMovingTimeoutManager.register(stEventEntity := TC_EVENTS.OperationalErrors2.Y2StartMoveUpTimeout, timerTime := T#1S, conformation := TRUE, sensorID := sensorID_t.EXPANTION_SENSOR_B2_Y2_UP, actorID := actorID_t.ACTOR_Y2_OUT, expectedActorValue := TRUE, waitHWConformation := FALSE);
_actorStartMovingTimeoutManager.register(stEventEntity := TC_EVENTS.OperationalErrors2.Y3StartMoveDownTimeout, timerTime := T#1S, conformation := TRUE, sensorID := sensorID_t.SENSOR_B3_Y3_DOWN, actorID := actorID_t.ACTOR_Y3_OUT, expectedActorValue := FALSE, waitHWConformation := FALSE);
_actorStartMovingTimeoutManager.register(stEventEntity := TC_EVENTS.OperationalErrors2.Y3StartMoveUpTimeout, timerTime := T#1S, conformation := TRUE, sensorID := sensorID_t.SENSOR_B4_Y3_UP, actorID := actorID_t.ACTOR_Y3_OUT, expectedActorValue := TRUE, waitHWConformation := FALSE);

_primitiveWatchdogManager.register(stEventEntity := TC_EVENTS.OperationalErrors2.LowPneumaticPressure, timerTime := T#10S, conformation := TRUE, sensorID := sensorID_t.SENSOR_PNEUMATIC_PRESHURE_OK, waitHWConformation := FALSE);
_primitiveWatchdogManager.register(stEventEntity := TC_EVENTS.OperationalErrors.EmStopPressed, timerTime := T#100MS, conformation := TRUE, sensorPtr := ADR(InputOutput.EmStop), waitHWConformation := FALSE);

_IOExpantionMessageErrorHandler.register(stEventEntity := TC_EVENTS.ProgrammingErrors.testError, timerTime := T#10MS, conformation := TRUE, diagCodeErrorMessage := diagCodeErrorTestMessage, textIDErrorMessage := textIDErrorTestMessage, diagCodeClearMessage := diagCodeClearTestMessage, textIDClearMessage := textIDClearTestMessage);
END_METHOD

// resets all errors 
METHOD reset : BOOL
VAR_INPUT
END_VAR
_actorMovingTimeoutManager.resetAll();
_actorStartMovingTimeoutManager.resetAll();
_primitiveWatchdogManager.resetAll();
_IOExpantionMessageErrorHandler.resetAll();
END_METHOD

METHOD setIOExpantionHandler : BOOL
VAR_INPUT
	IOExpantionHandlerPtr : POINTER TO IOExpantionHandler_t;
END_VAR
_IOExpantionHandler := IOExpantionHandlerPtr;
_actorMovingTimeoutManager.setIOExpantionHandler(_IOExpantionHandler);
_actorStartMovingTimeoutManager.setIOExpantionHandler(_IOExpantionHandler);
_primitiveWatchdogManager.setIOExpantionHandler(_IOExpantionHandler);
_IOExpantionMessageErrorHandler.setIOExpantionHandler(_IOExpantionHandler);

setIOExpantionHandler := TRUE;
return;
END_METHOD

METHOD startErrors : BOOL
VAR_INPUT
END_VAR
THIS^._trowErrors := TRUE;

startErrors := TRUE;
RETURN;
END_METHOD

METHOD stopErrors : BOOL
VAR_INPUT
END_VAR
THIS^._trowErrors := False;

stopErrors := TRUE;
RETURN;
END_METHOD

// call this method every sycle
METHOD update : BOOL
VAR_INPUT
END_VAR
IF _IOExpantionHandler = NULL THEN
	update := FALSE;
	RETURN;
END_IF

IF _errorsInitialised = FALSE THEN
	initErrors();
	_errorsInitialised := TRUE;
END_IF

// is not an actor error and can appear outside of opperations.
//_IOExpantionMessageErrorHandler.update(); 
{warning 'disabled IOExpantionMessageErrorHandler'}

IF _trowErrors = FALSE THEN
	update := TRUE;
	RETURN;
END_IF

_actorMovingTimeoutManager.update();
_actorStartMovingTimeoutManager.update();
_primitiveWatchdogManager.update();

update := TRUE;
RETURN;
END_METHOD

END_FUNCTION_BLOCK

// ---- POUs/ErrorSystem/ActorMovingTimeoutManager_t.TcPOU
{attribute 'enable_dynamic_creation'}
FUNCTION_BLOCK ActorMovingTimeoutManager_t
VAR_INPUT
END_VAR
VAR_OUTPUT
END_VAR
VAR
	_actorMovingTimeoutArray : ARRAY [0..99] OF  ActorMovingTimeoutEx_t;
	_maxActorMovingTimeoutIndex : UINT := 99;
	_currentActorMovingTimeoutIndex : UINT := 0;
	_ErrorMessage : FB_TcMessage;
	_IOExpantionHandler : POINTER TO IOExpantionHandler_t := NULL;
	
	_IOExpantionHandlerNotValidErrorSent : BOOL := FALSE;
END_VAR

// clears and destroyes all AcrtorMovingTimeouts
METHOD clear : BOOL
VAR_INPUT
END_VAR

VAR
	i: UINT;
END_VAR
_currentActorMovingTimeoutIndex := 0;

clear := TRUE;
RETURN;
END_METHOD

// confirm all ActorMovingTimeouts
METHOD confirmAll : BOOL
VAR_INPUT
END_VAR

VAR
	i: UINT;
END_VAR
// confirm all alarms
FOR i := 0 TO _currentActorMovingTimeoutIndex DO
	_actorMovingTimeoutArray[i].ActorMovingTimeout.confirm();
END_FOR

confirmAll := TRUE;
RETURN;
END_METHOD

METHOD hasError : BOOL
VAR_INPUT
END_VAR

VAR
	i: UINT;
END_VAR
FOR i := 0 TO _currentActorMovingTimeoutIndex DO
	hasError := hasError OR THIS^._actorMovingTimeoutArray[i].ActorMovingTimeout.isAlarmRaised();
END_FOR

RETURN;
END_METHOD

// register a ActorMovingTimeout
METHOD register : BOOL
VAR_INPUT
	stEventEntity : TcEventEntry;
	timerTime : TIME; // sets the timer for the timeout
	conformation : BOOL := TRUE; 
	waitHWConformation : bool := true;
	sensor1 : POINTER TO BOOL := NULL;
	sensor2 : POINTER TO BOOL := NULL;
	sensor3 : POINTER TO BOOL := NULL;
	sensorID1 : sensorID_t := sensorID_t.SENSOR_NO_SENSOR;
	sensorID2 : sensorID_t := sensorID_t.SENSOR_NO_SENSOR;
	sensorID3 : sensorID_t := sensorID_t.SENSOR_NO_SENSOR;
END_VAR

VAR
	_tmpStr: STRING;
END_VAR
IF _currentActorMovingTimeoutIndex + 1 > _maxActorMovingTimeoutIndex THEN
	_ErrorMessage.CreateEx(TC_EVENTS.ProgrammingErrors.ExceedingAllowedAmountOfActorMovingTimeoutTimeouts, 0 );
	_ErrorMessage.ipArguments.AddString(__POUNAME());
	_tmpStr := formatPosition(__POSITION());
	_ErrorMessage.ipArguments.AddString(_tmpStr);
	_ErrorMessage.ipArguments.AddUInt(_maxActorMovingTimeoutIndex);
	_ErrorMessage.Send(0);
	
	register := FALSE;
	RETURN;
END_IF

IF sensor1 = NULL AND sensor2 = NULL AND sensor3 = NULL AND sensorID1 = sensorID_t.SENSOR_NO_SENSOR AND sensorID2 = sensorID_t.SENSOR_NO_SENSOR AND sensorID3 = sensorID_t.SENSOR_NO_SENSOR THEN
	_ErrorMessage.CreateEx(TC_EVENTS.ProgrammingErrors.ActorMovingTimeoutNoValidSensorGiven, 0 );
	_ErrorMessage.ipArguments.AddString(__POUNAME());
	_tmpStr := formatPosition(__POSITION());
	_ErrorMessage.ipArguments.AddString(_tmpStr);
	_ErrorMessage.Send(0);
	
	register := FALSE;
	RETURN;
END_IF

_currentActorMovingTimeoutIndex := _currentActorMovingTimeoutIndex + 1; // increase it by one

_actorMovingTimeoutArray[_currentActorMovingTimeoutIndex].ActorMovingTimeout.register(stEventEntity, timerTime, conformation, waitHWConformation);
_actorMovingTimeoutArray[_currentActorMovingTimeoutIndex].sensorPtr1 := sensor1;
_actorMovingTimeoutArray[_currentActorMovingTimeoutIndex].sensorPtr2 := sensor2;
_actorMovingTimeoutArray[_currentActorMovingTimeoutIndex].sensorPtr3 := sensor3;
_actorMovingTimeoutArray[_currentActorMovingTimeoutIndex].sensorID1 := sensorID1;
_actorMovingTimeoutArray[_currentActorMovingTimeoutIndex].sensorID2 := sensorID2;
_actorMovingTimeoutArray[_currentActorMovingTimeoutIndex].sensorID3 := sensorID3;

register := TRUE;
RETURN;
END_METHOD

// reset all ActorMovingTimeoutos
METHOD resetAll : BOOL
VAR_INPUT
END_VAR

VAR
	i: UINT;
END_VAR
// confirm all alarms
FOR i := 0 TO _currentActorMovingTimeoutIndex DO
	_actorMovingTimeoutArray[i].ActorMovingTimeout.reset();
END_FOR

resetAll := TRUE;
RETURN;
END_METHOD

// resolvs the status of the sensors
METHOD PRIVATE resolveSensors : BOOL
VAR_INPUT
	ActorMovingTimeoutEx : ActorMovingTimeoutEx_t;
END_VAR

VAR
	_tmpStr: STRING;
	_sensor: BOOL;
END_VAR
IF _IOExpantionHandler = NULL AND _IOExpantionHandlerNotValidErrorSent = FALSE THEN
	_IOExpantionHandlerNotValidErrorSent := TRUE;
	_ErrorMessage.CreateEx(TC_EVENTS.ProgrammingErrors.NoValidPointerToIOExpantionHandler, 0 );
	_ErrorMessage.ipArguments.AddString(__POUNAME());
	_tmpStr := formatPosition(__POSITION());
	_ErrorMessage.ipArguments.AddString(_tmpStr);
	_ErrorMessage.ipArguments.AddUInt(_maxActorMovingTimeoutIndex);
	_ErrorMessage.Send(0);
END_IF

IF ActorMovingTimeoutEx.sensorPtr1 <> NULL THEN
	_sensor := _sensor OR ActorMovingTimeoutEx.sensorPtr1^;
END_IF

IF ActorMovingTimeoutEx.sensorPtr2 <> NULL THEN
	_sensor := _sensor OR ActorMovingTimeoutEx.sensorPtr2^;
END_IF

IF ActorMovingTimeoutEx.sensorPtr3 <> NULL THEN
	_sensor := _sensor OR ActorMovingTimeoutEx.sensorPtr3^;
END_IF 

// no IOExpantionHandler
IF _IOExpantionHandler = NULL THEN 
	resolveSensors := _sensor;
	RETURN;
END_IF

IF ActorMovingTimeoutEx.sensorID1 <> sensorID_t.SENSOR_NO_SENSOR THEN
	_sensor := _sensor OR _IOExpantionHandler^.getSensorStatus(ActorMovingTimeoutEx.sensorID1);
END_IF

IF ActorMovingTimeoutEx.sensorID2 <> sensorID_t.SENSOR_NO_SENSOR THEN
	_sensor := _sensor OR _IOExpantionHandler^.getSensorStatus(ActorMovingTimeoutEx.sensorID2);
END_IF

IF ActorMovingTimeoutEx.sensorID3 <> sensorID_t.SENSOR_NO_SENSOR THEN
	_sensor := _sensor OR _IOExpantionHandler^.getSensorStatus(ActorMovingTimeoutEx.sensorID3);
END_IF

resolveSensors := _sensor;
RETURN;
END_METHOD

// sets the IOExpantionHandler refferance
METHOD setIOExpantionHandler : BOOL
VAR_INPUT
	IOExpantionHandlerPtr : POINTER TO IOExpantionHandler_t;
END_VAR
_IOExpantionHandler := IOExpantionHandlerPtr;
setIOExpantionHandler := TRUE;
RETURN;
END_METHOD

// update all ActorMovingTimeout, call this every cycle
METHOD update : BOOL
VAR_INPUT
END_VAR

VAR
	i: UINT;
	_sensor : bool := false;
END_VAR
FOR i := 0 TO _currentActorMovingTimeoutIndex DO
	_actorMovingTimeoutArray[i].ActorMovingTimeout.update(resolveSensors(_actorMovingTimeoutArray[i]));
END_FOR

update := TRUE;
RETURN;
END_METHOD

END_FUNCTION_BLOCK

// ---- POUs/ErrorSystem/ActorStartMovingTimeoutManager_t.TcPOU
FUNCTION_BLOCK ActorStartMovingTimeoutManager_t
VAR_INPUT
END_VAR
VAR_OUTPUT
END_VAR
VAR
	_actorStartMovingTimeoutArray : ARRAY [0..99] OF  ActorStartMovingtimeoutEx_t;
	_maxActorStartMovingTimeoutIndex : UINT := 99;
	_currentActorStartMovingTimeoutIndex : UINT := 0;
	_ErrorMessage : FB_TcMessage;
	_IOExpantionHandler : POINTER TO IOExpantionHandler_t := NULL;
	
	_IOExpantionHandlerNotValidErrorSent : BOOL := FALSE;
END_VAR

// clears and destroyes all AcrtorStartMovingTimeouts
METHOD clear : BOOL
VAR_INPUT
END_VAR
_currentActorStartMovingTimeoutIndex := 0;

clear := TRUE;
RETURN;
END_METHOD

// confirm all ActorStartMovingTimeouts
METHOD confirmAll : BOOL
VAR_INPUT
END_VAR

VAR
	i : UINT;
END_VAR
// confirm all alarms
FOR i := 0 TO _currentActorStartMovingTimeoutIndex DO
	_actorStartMovingTimeoutArray[i].ActorStartMovingTimeout.confirm();
END_FOR

confirmAll := TRUE;
RETURN;
END_METHOD

// if true an error has been trown
METHOD hasError : BOOL
VAR_INPUT
END_VAR
VAR
	i : UINT := 0;
END_VAR
FOR i := 0 TO _currentActorStartMovingTimeoutIndex DO
	hasError := hasError OR THIS^._actorStartMovingTimeoutArray[i].ActorStartMovingTimeout.isAlarmRaised();
END_FOR

RETURN;
END_METHOD

METHOD register : BOOL
VAR_INPUT
	stEventEntity : TcEventEntry;
	timerTime : TIME; // sets the timer for the timeout
	conformation : BOOL := TRUE; 
	expectedActorValue : BOOL; // actor value when sensor is true
	sensorPtr : POINTER TO BOOL := NULL; 
	actorPtr : POINTER TO BOOL := NULL;
	sensorID : sensorID_t := sensorID_t.SENSOR_NO_SENSOR;
	actorID : actorID_t := actorID_t.ACTOR_NO_ACTOR;
	waitHWConformation : BOOL := TRUE;
END_VAR

VAR
	_tmpStr: STRING;
END_VAR
IF _currentActorStartMovingTimeoutIndex + 1 > _maxActorStartMovingTimeoutIndex THEN
	_ErrorMessage.CreateEx(TC_EVENTS.ProgrammingErrors.ExceedingAllowedAmountOfActorMovingTimeoutTimeouts, 0 );
	_ErrorMessage.ipArguments.AddString(__POUNAME());
	_tmpStr := formatPosition(__POSITION());
	_ErrorMessage.ipArguments.AddString(_tmpStr);
	_ErrorMessage.ipArguments.AddUInt(_maxActorStartMovingTimeoutIndex);
	_ErrorMessage.Send(0);
	
	register := FALSE;
	RETURN;
END_IF

IF (NOT (sensorPtr = NULL XOR sensorID = sensorID_t.SENSOR_NO_SENSOR)) OR ( NOT (actorPtr = NULL XOR actorID = actorID_t.ACTOR_NO_ACTOR)) THEN
	_ErrorMessage.CreateEx(TC_EVENTS.ProgrammingErrors.ActorMovingTimeoutNoValidSensorGiven, 0 );
	_ErrorMessage.ipArguments.AddString(__POUNAME());
	_tmpStr := formatPosition(__POSITION());
	_ErrorMessage.ipArguments.AddString(_tmpStr);
	_ErrorMessage.Send(0);
	
	register := FALSE;
	RETURN;
END_IF

_currentActorStartMovingTimeoutIndex := _currentActorStartMovingTimeoutIndex + 1; // increase it by one

